KUKA KRL program: Up86.src, Up86.dat

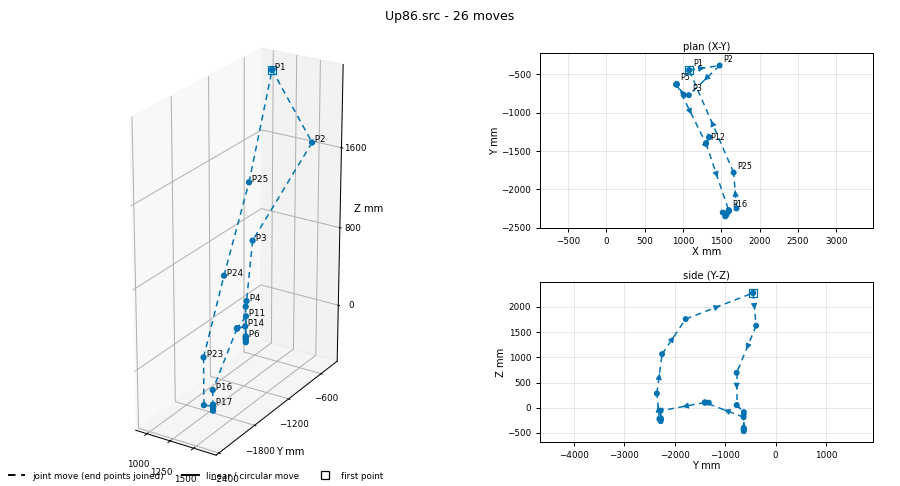
[picture p0: tool path of Up86.src, 26 of 26 moves have a stored position in this frame; points joined in program order, loops and branches not executed]
--- Up86.src ---
&ACCESS RVP
&REL 328
&COMMENT Abdocken 380 Andocken 379
&PARAM DISKPATH = KRC:\R1\UPs
&PARAM TEMPLATE = C:\KRC\Roboter\Template\upvorgabe
&PARAM EDITMASK = Up999[1-999]
&PARAM TPVW_VERSION = 8.1.8
DEF UP86()
   ; FOLD UP Anfang;%{SE} %MKUKATPVW
   SPS_N=-1
   SPS_FERTIG=FALSE
   IF NOT CALLBYSELECT THEN
      INTERRUPT DECL 10 WHEN $CYCFLAG[254]==FALSE DO VW(#FB_STOP,TRUE)
      INTERRUPT ON 10
      INT10=TRUE
      VW_USR_R (#USR_INIT)
   ENDIF
   VW(#VW_INIT_UP,TRUE)
   ; ENDFOLD
   ;FOLD -- TUHR Roboter 5475R01 -- ;%{PSE}%MKUKATPVW,%CVW_COM,%VCOMMENT,%P 1:Comment:, 2:TUHR Roboter 5475R01
      ;FOLD {H}
         M_COMMENT("TUHR Roboter 5475R01")
      ;ENDFOLD
   ;ENDFOLD
   ;FOLD -- Abdocken  VW380 Andocken VW379 -- ;%{PSE}%MKUKATPVW,%CVW_COM,%VCOMMENT,%P 1:Comment:, 2:Abdocken  VW380 Andocken VW379
      ;FOLD {H}
         M_COMMENT("Abdocken  VW380 Andocken VW379")
      ;ENDFOLD
   ;ENDFOLD
   ;FOLD -- DB1 Abdeckklappe AUF -- ;%{PSE}%MKUKATPVW,%CVW_COM,%VCOMMENT,%P 1:Comment:, 2:DB1 Abdeckklappe AUF
      ;FOLD {H}
         M_COMMENT("DB1 Abdeckklappe AUF")
      ;ENDFOLD
   ;ENDFOLD
   ;FOLD -- DB2 Abdeckklappe AUF -- ;%{PSE}%MKUKATPVW,%CVW_COM,%VCOMMENT,%P 1:Comment:, 2:DB2 Abdeckklappe AUF
      ;FOLD {H}
         M_COMMENT("DB2 Abdeckklappe AUF")
      ;ENDFOLD
   ;ENDFOLD
   ;FOLD -- Gespert nur 1 Greifer vorhanden -- ;%{PSE}%MKUKATPVW,%CVW_COM,%VCOMMENT,%P 1:Comment:, 2:Gespert nur 1 Greifer vorhanden
      ;FOLD {H}
         M_COMMENT("Gespert nur 1 Greifer vorhanden")
      ;ENDFOLD
   ;ENDFOLD
   ;FOLD PTP VB=100% VE=0% ACC=100% RobWzg=32 Base=0 SPSTrig=0[1/100s] P ;%{P}%MKUKATPVW,%CMOVE8,%VPTP,%P 1:1, 2: VB=, 3:100, 4:%, 5: VE=, 6:0, 7:%, 8: ACC=, 9:100, 10:%, 11: RobWzg=, 12:32, 13: Base=, 14:0, 15: SPSTrig=, 16:0, 17:[1/100s], 18: P, 19:1, 20:-1, 21:1
      ;FOLD 1: FB PSPS = AUS ;%{SE}%MKUKATPVW %CVW_SPS %VFBPSPS %P 2:FB PSPS = AUS,3:FBPSPS
      ;ENDFOLD
      ;FOLD 2: A23 = AUS ;%{SE}%MKUKATPVW %CVW_SPS %VBOASG %P 2:A23 = AUS,3:BOASG
      ;ENDFOLD
      ;FOLD 3: t6 ( EIN ) = 0[1/10Sek] ;%{SE}%MKUKATPVW %CVW_SPS %VTASG %P 2:t6 ( EIN ) = 0[1/10Sek],3:TASG
      ;ENDFOLD
      ;FOLD 4: SPSMAKRO50 = EIN ;%{SE}%MKUKATPVW %CVW_SPS %VMAKRO %P 2:SPSMAKRO50 = EIN,3:MAKRO
      ;ENDFOLD
      ;FOLD 5: SPSMAKRO53 = EIN ;%{SE}%MKUKATPVW %CVW_SPS %VMAKRO %P 2:SPSMAKRO53 = EIN,3:MAKRO
      ;ENDFOLD
      ;FOLD 6: A42 = EIN ;%{SE}%MKUKATPVW %CVW_SPS %VBOASG %P 2:A42 = EIN,3:BOASG
      ;ENDFOLD
      ;FOLD 7: A43 = EIN ;%{SE}%MKUKATPVW %CVW_SPS %VBOASG %P 2:A43 = EIN,3:BOASG
      ;ENDFOLD
      ;FOLD 8: A44 = EIN ;%{SE}%MKUKATPVW %CVW_SPS %VBOASG %P 2:A44 = EIN,3:BOASG
      ;ENDFOLD
      ;FOLD 9: A45 = EIN ;%{SE}%MKUKATPVW %CVW_SPS %VBOASG %P 2:A45 = EIN,3:BOASG
      ;ENDFOLD
      ;FOLD 10: A47 = EIN ;%{SE}%MKUKATPVW %CVW_SPS %VBOASG %P 2:A47 = EIN,3:BOASG
      ;ENDFOLD
      ;FOLD 11: A49 = EIN ;%{SE}%MKUKATPVW %CVW_SPS %VBOASG %P 2:A49 = EIN,3:BOASG
      ;ENDFOLD
      ;FOLD 12: A52 = EIN ;%{SE}%MKUKATPVW %CVW_SPS %VBOASG %P 2:A52 = EIN,3:BOASG
      ;ENDFOLD
      ;FOLD 13: A54 = EIN ;%{SE}%MKUKATPVW %CVW_SPS %VBOASG %P 2:A54 = EIN,3:BOASG
      ;ENDFOLD
      ;FOLD 14: A75 = EIN ;%{SE}%MKUKATPVW %CVW_SPS %VBOASG %P 2:A75 = EIN,3:BOASG
      ;ENDFOLD
      ;FOLD 15: A76 = EIN ;%{SE}%MKUKATPVW %CVW_SPS %VBOASG %P 2:A76 = EIN,3:BOASG
      ;ENDFOLD
      ;FOLD 16: A79 = EIN ;%{SE}%MKUKATPVW %CVW_SPS %VBOASG %P 2:A79 = EIN,3:BOASG
      ;ENDFOLD
      ;FOLD 17: A80 = EIN ;%{SE}%MKUKATPVW %CVW_SPS %VBOASG %P 2:A80 = EIN,3:BOASG
      ;ENDFOLD
      ;FOLD 18: WARTE BIS M13 & M78 & !E16 ;%{SE}%MKUKATPVW %CVW_SPS %VWBOASG %P 2:WARTE BIS M13 & M78 & !E16,3:WBOASG
      ;ENDFOLD
      ;FOLD 19: F1 = EIN ;%{SE}%MKUKATPVW %CVW_SPS %VBOASG %P 2:F1 = EIN,3:BOASG
      ;ENDFOLD
      ;FOLD 20: F2 = EIN ;%{SE}%MKUKATPVW %CVW_SPS %VBOASG %P 2:F2 = EIN,3:BOASG
      ;ENDFOLD
      ;FOLD 21: SPSMAKRO343 = M13 ;%{SE}%MKUKATPVW %CVW_SPS %VMAKRO %P 2:SPSMAKRO343 = M13,3:MAKRO
      ;ENDFOLD
      ;FOLD 22: SPSMAKRO340 = EIN ;%{SE}%MKUKATPVW %CVW_SPS %VMAKRO %P 2:SPSMAKRO340 = EIN,3:MAKRO
      ;ENDFOLD
      ;FOLD 23: WARTE BIS M32 & M34 ;%{SE}%MKUKATPVW %CVW_SPS %VWBOASG %P 2:WARTE BIS M32 & M34,3:WBOASG
      ;ENDFOLD
      ;FOLD 24: SPSMAKRO430 = EIN ;%{SE}%MKUKATPVW %CVW_SPS %VMAKRO %P 2:SPSMAKRO430 = EIN,3:MAKRO
      ;ENDFOLD
      ;FOLD 25: F841 = EIN ;%{SE}%MKUKATPVW %CVW_SPS %VBOASG %P 2:F841 = EIN,3:BOASG
      ;ENDFOLD
      ;FOLD 26: F842 = EIN ;%{SE}%MKUKATPVW %CVW_SPS %VBOASG %P 2:F842 = EIN,3:BOASG
      ;ENDFOLD
      ;FOLD 27: SPSMAKRO432 = EIN ;%{SE}%MKUKATPVW %CVW_SPS %VMAKRO %P 2:SPSMAKRO432 = EIN,3:MAKRO
      ;ENDFOLD
      ;FOLD 28: WARTE BIS E547 & !E548 & E549 & !E550 & E552 ;%{SE}%MKUKATPVW %CVW_SPS %VWBOASG %P 2:WARTE BIS E547 & !E548 & E549 & !E550 & E552,3:WBOASG
      ;ENDFOLD
      ;FOLD 29: WARTE BIS E23 ;%{SE}%MKUKATPVW %CVW_SPS %VWBOASG %P 2:WARTE BIS E23,3:WBOASG
      ;ENDFOLD
      ;FOLD 30: A23 = EIN ;%{SE}%MKUKATPVW %CVW_SPS %VBOASG %P 2:A23 = EIN,3:BOASG
      ;ENDFOLD
      ;FOLD 31: FB PSPS = M30 & M32 & M34 & M78 & M82 & E547 & E549 ;%{SE}%MKUKATPVW %CVW_SPS %VFBPSPS %P 2:FB PSPS = M30 & M32 & M34 & M78 & M82 & E547 & E549,3:FBPSPS
      ;ENDFOLD
      ;FOLD {H}
         VW_MPARA_ACT=P1_D
         Act_P1 = P1
         Act_P2 = P1
         VW(#MPARA,TRUE)
         SPS_FERTIG=FALSE
         TRIGGER WHEN DISTANCE=1 DELAY=0 DO SPS_TRIG(1) PRIO=-1
         PTP P1
         $ADVANCE=1
         WAIT FOR SPS_FERTIG
      ;ENDFOLD
   ;ENDFOLD
   ;FOLD PTP VB=100% VE=100% ACC=100% RobWzg=32 Base=0 SPSTrig=0[1/100s] P ;%{P}%MKUKATPVW,%CMOVE8,%VPTP,%P 1:1, 2: VB=, 3:100, 4:%, 5: VE=, 6:100, 7:%, 8: ACC=, 9:100, 10:%, 11: RobWzg=, 12:32, 13: Base=, 14:0, 15: SPSTrig=, 16:0, 17:[1/100s], 18: P, 19:2, 20:-1, 21:2
      ;FOLD 1: FB PSPS = M30 & M32 & M34 & M78 & M82 & E547 & E549 ;%{SE}%MKUKATPVW %CVW_SPS %VFBPSPS %P 2:FB PSPS = M30 & M32 & M34 & M78 & M82 & E547 & E549,3:FBPSPS
      ;ENDFOLD
      ;FOLD {H}
         VW_MPARA_ACT=P2_D
         Act_P1 = P2
         Act_P2 = P2
         VW(#MPARA,TRUE)
         SPS_FERTIG=FALSE
         TRIGGER WHEN DISTANCE=1 DELAY=0 DO SPS_TRIG(10002) PRIO=-1
         PTP P2 C_PTP C_VEL
         $ADVANCE=1
      ;ENDFOLD
   ;ENDFOLD
   ;FOLD PTP VB=100% VE=100% ACC=100% RobWzg=32 Base=0 SPSTrig=0[1/100s] P ;%{P}%MKUKATPVW,%CMOVE8,%VPTP,%P 1:1, 2: VB=, 3:100, 4:%, 5: VE=, 6:100, 7:%, 8: ACC=, 9:100, 10:%, 11: RobWzg=, 12:32, 13: Base=, 14:0, 15: SPSTrig=, 16:0, 17:[1/100s], 18: P, 19:3, 20:-1, 21:3
      ;FOLD 1: FB PSPS = M30 & M32 & M34 & M78 & M82 & E547 & E549 ;%{SE}%MKUKATPVW %CVW_SPS %VFBPSPS %P 2:FB PSPS = M30 & M32 & M34 & M78 & M82 & E547 & E549,3:FBPSPS
      ;ENDFOLD
      ;FOLD {H}
         VW_MPARA_ACT=P3_D
         Act_P1 = P3
         Act_P2 = P3
         VW(#MPARA,TRUE)
         SPS_FERTIG=FALSE
         TRIGGER WHEN DISTANCE=1 DELAY=0 DO SPS_TRIG(10003) PRIO=-1
         PTP P3 C_PTP C_VEL
         $ADVANCE=1
      ;ENDFOLD
   ;ENDFOLD
   ;FOLD PTP VB=100% VE=100% ACC=100% RobWzg=32 Base=0 SPSTrig=0[1/100s] P ;%{P}%MKUKATPVW,%CMOVE8,%VPTP,%P 1:1, 2: VB=, 3:100, 4:%, 5: VE=, 6:100, 7:%, 8: ACC=, 9:100, 10:%, 11: RobWzg=, 12:32, 13: Base=, 14:0, 15: SPSTrig=, 16:0, 17:[1/100s], 18: P, 19:4, 20:-1, 21:4
      ;FOLD 1: FB PSPS = M30 & M32 & M34 & M78 & M82 & E547 & E549 ;%{SE}%MKUKATPVW %CVW_SPS %VFBPSPS %P 2:FB PSPS = M30 & M32 & M34 & M78 & M82 & E547 & E549,3:FBPSPS
      ;ENDFOLD
      ;FOLD {H}
         VW_MPARA_ACT=P4_D
         Act_P1 = P4
         Act_P2 = P4
         VW(#MPARA,TRUE)
         SPS_FERTIG=FALSE
         TRIGGER WHEN DISTANCE=1 DELAY=0 DO SPS_TRIG(10004) PRIO=-1
         PTP P4 C_PTP C_VEL
         $ADVANCE=1
      ;ENDFOLD
   ;ENDFOLD
   ;FOLD PTP VB=100% VE=100% ACC=100% RobWzg=32 Base=0 SPSTrig=0[1/100s] P ;%{P}%MKUKATPVW,%CMOVE8,%VPTP,%P 1:1, 2: VB=, 3:100, 4:%, 5: VE=, 6:100, 7:%, 8: ACC=, 9:100, 10:%, 11: RobWzg=, 12:32, 13: Base=, 14:0, 15: SPSTrig=, 16:0, 17:[1/100s], 18: P, 19:5, 20:-1, 21:5
      ;FOLD 1: FB PSPS = M30 & M32 & M34 & M78 & M82 & E547 & E549 ;%{SE}%MKUKATPVW %CVW_SPS %VFBPSPS %P 2:FB PSPS = M30 & M32 & M34 & M78 & M82 & E547 & E549,3:FBPSPS
      ;ENDFOLD
      ;FOLD {H}
         VW_MPARA_ACT=P5_D
         Act_P1 = P5
         Act_P2 = P5
         VW(#MPARA,TRUE)
         SPS_FERTIG=FALSE
         TRIGGER WHEN DISTANCE=1 DELAY=0 DO SPS_TRIG(10005) PRIO=-1
         PTP P5 C_PTP C_VEL
         $ADVANCE=1
      ;ENDFOLD
   ;ENDFOLD
   ;FOLD -- Profinet  Teilnehmer  abschalten -- ;%{PSE}%MKUKATPVW,%CVW_COM,%VCOMMENT,%P 1:Comment:, 2:Profinet  Teilnehmer  abschalten
      ;FOLD {H}
         M_COMMENT("Profinet  Teilnehmer  abschalten")
      ;ENDFOLD
   ;ENDFOLD
   ;FOLD PTP VB=100% VE=0% ACC=100% RobWzg=32 Base=0 SPSTrig=0[1/100s] P ;%{P}%MKUKATPVW,%CMOVE8,%VPTP,%P 1:1, 2: VB=, 3:100, 4:%, 5: VE=, 6:0, 7:%, 8: ACC=, 9:100, 10:%, 11: RobWzg=, 12:32, 13: Base=, 14:0, 15: SPSTrig=, 16:0, 17:[1/100s], 18: P, 19:6, 20:-1, 21:6
      ;FOLD 1: FB PSPS = EIN ;%{SE}%MKUKATPVW %CVW_SPS %VFBPSPS %P 2:FB PSPS = EIN,3:FBPSPS
      ;ENDFOLD
      ;FOLD 2: A23 = AUS ;%{SE}%MKUKATPVW %CVW_SPS %VBOASG %P 2:A23 = AUS,3:BOASG
      ;ENDFOLD
      ;FOLD 3: SPSMAKRO422 = !E540 ;%{SE}%MKUKATPVW %CVW_SPS %VMAKRO %P 2:SPSMAKRO422 = !E540,3:MAKRO
      ;ENDFOLD
      ;FOLD 4: WARTE BIS E540 & !E551 & E23 ;%{SE}%MKUKATPVW %CVW_SPS %VWBOASG %P 2:WARTE BIS E540 & !E551 & E23,3:WBOASG
      ;ENDFOLD
      ;FOLD 5: TECH3_ PN-Docken ID-Nr =122 Abschalten EIN ;%{SE}%MKUKATPVW %CVW_SPS %VUSER %P 2:TECH3_.PN-Docken P1= 122 P2= 60 P3= 1 P4= 1 P5= 1 P6= 1 P7=EIN P8=301,3:USER
      ;ENDFOLD
      ;FOLD 6: A23 = EIN ;%{SE}%MKUKATPVW %CVW_SPS %VBOASG %P 2:A23 = EIN,3:BOASG
      ;ENDFOLD
      ;FOLD 7: FB PSPS = M30 & M78 & E547 & E549 ;%{SE}%MKUKATPVW %CVW_SPS %VFBPSPS %P 2:FB PSPS = M30 & M78 & E547 & E549,3:FBPSPS
      ;ENDFOLD
      ;FOLD {H}
         VW_MPARA_ACT=P6_D
         Act_P1 = P6
         Act_P2 = P6
         VW(#MPARA,TRUE)
         SPS_FERTIG=FALSE
         TRIGGER WHEN DISTANCE=1 DELAY=0 DO SPS_TRIG(6) PRIO=-1
         VW_USER (#USR_ADV,301,122,60,1,1,1,1,TRUE)
         VW_USR_R (#USR_ADV,301,122,60,1,1,1,1,TRUE)
         PTP P6
         $ADVANCE=1
         WAIT FOR SPS_FERTIG
         VW_USER (#USR_MAIN,301,122,60,1,1,1,1,TRUE)
         VW_USR_R (#USR_MAIN,301,122,60,1,1,1,1,TRUE)
      ;ENDFOLD
   ;ENDFOLD
   ;FOLD -- Ueber  DB -- ;%{PSE}%MKUKATPVW,%CVW_COM,%VCOMMENT,%P 1:Comment:, 2:Ueber  DB
      ;FOLD {H}
         M_COMMENT("Ueber  DB")
      ;ENDFOLD
   ;ENDFOLD
   ;FOLD LIN VB=200[mm/s] VE=0% ACC=100% RobWzg=32 Base=0 SPSTrig=5[1/100s] P ;%{P}%MKUKATPVW,%CMOVE8,%VLIN,%P 1:2, 2: VB=, 3:200, 4:[mm/s], 5: VE=, 6:0, 7:%, 8: ACC=, 9:100, 10:%, 11: RobWzg=, 12:32, 13: Base=, 14:0, 15: SPSTrig=, 16:5, 17:[1/100s], 18: P, 19:7, 20:-1, 21:7
      ;FOLD 1: FB PSPS = M30 & M78 & E547 & E549 ;%{SE}%MKUKATPVW %CVW_SPS %VFBPSPS %P 2:FB PSPS = M30 & M78 & E547 & E549,3:FBPSPS
      ;ENDFOLD
      ;FOLD {H}
         VW_MPARA_ACT=P7_D
         Act_P1 = P7
         Act_P2 = P7
         VW(#MPARA,TRUE)
         SPS_FERTIG=FALSE
         TRIGGER WHEN DISTANCE=1 DELAY=-50 DO SPS_TRIG(7) PRIO=-1
         LIN P7
         $ADVANCE=1
         WAIT FOR SPS_FERTIG
      ;ENDFOLD
   ;ENDFOLD
   ;FOLD -- Abdockposition VW380 4T 5425r01 -- ;%{PSE}%MKUKATPVW,%CVW_COM,%VCOMMENT,%P 1:Comment:, 2:Abdockposition VW380 4T 5425r01
      ;FOLD {H}
         M_COMMENT("Abdockposition VW380 4T 5425r01")
      ;ENDFOLD
   ;ENDFOLD
   ;FOLD LIN VB=50[mm/s] VE=0% ACC=100% RobWzg=32 Base=0 SPSTrig=5[1/100s] P ;%{P}%MKUKATPVW,%CMOVE8,%VLIN,%P 1:2, 2: VB=, 3:50, 4:[mm/s], 5: VE=, 6:0, 7:%, 8: ACC=, 9:100, 10:%, 11: RobWzg=, 12:32, 13: Base=, 14:0, 15: SPSTrig=, 16:5, 17:[1/100s], 18: P, 19:8, 20:-1, 21:8
      ;FOLD 1: FB PSPS = EIN ;%{SE}%MKUKATPVW %CVW_SPS %VFBPSPS %P 2:FB PSPS = EIN,3:FBPSPS
      ;ENDFOLD
      ;FOLD 2: A23 = AUS ;%{SE}%MKUKATPVW %CVW_SPS %VBOASG %P 2:A23 = AUS,3:BOASG
      ;ENDFOLD
      ;FOLD 3: WARTE BIS E540 & E551 & E23 ;%{SE}%MKUKATPVW %CVW_SPS %VWBOASG %P 2:WARTE BIS E540 & E551 & E23,3:WBOASG
      ;ENDFOLD
      ;FOLD 4: A23 = EIN ;%{SE}%MKUKATPVW %CVW_SPS %VBOASG %P 2:A23 = EIN,3:BOASG
      ;ENDFOLD
      ;FOLD 5: SPSMAKRO420 = EIN ;%{SE}%MKUKATPVW %CVW_SPS %VMAKRO %P 2:SPSMAKRO420 = EIN,3:MAKRO
      ;ENDFOLD
      ;FOLD 6: WARTE BIS !E538 & E539 ;%{SE}%MKUKATPVW %CVW_SPS %VWBOASG %P 2:WARTE BIS !E538 & E539,3:WBOASG
      ;ENDFOLD
      ;FOLD 7: FB PSPS = M30 & !E538 & E539 & E540 & E551 & E552 ;%{SE}%MKUKATPVW %CVW_SPS %VFBPSPS %P 2:FB PSPS = M30 & !E538 & E539 & E540 & E551 & E552,3:FBPSPS
      ;ENDFOLD
      ;FOLD {H}
         VW_MPARA_ACT=P8_D
         Act_P1 = P8
         Act_P2 = P8
         VW(#MPARA,TRUE)
         SPS_FERTIG=FALSE
         TRIGGER WHEN DISTANCE=1 DELAY=-50 DO SPS_TRIG(8) PRIO=-1
         LIN P8
         $ADVANCE=1
         WAIT FOR SPS_FERTIG
      ;ENDFOLD
   ;ENDFOLD
   ;FOLD -- Ueber  DB1  WASI  noch  belegt -- ;%{PSE}%MKUKATPVW,%CVW_COM,%VCOMMENT,%P 1:Comment:, 2:Ueber  DB1  WASI  noch  belegt
      ;FOLD {H}
         M_COMMENT("Ueber  DB1  WASI  noch  belegt")
      ;ENDFOLD
   ;ENDFOLD
   ;FOLD LIN VB=50[mm/s] VE=10% ACC=100% RobWzg=32 Base=0 SPSTrig=5[1/100s] P ;%{P}%MKUKATPVW,%CMOVE8,%VLIN,%P 1:2, 2: VB=, 3:50, 4:[mm/s], 5: VE=, 6:10, 7:%, 8: ACC=, 9:100, 10:%, 11: RobWzg=, 12:32, 13: Base=, 14:0, 15: SPSTrig=, 16:5, 17:[1/100s], 18: P, 19:9, 20:-1, 21:9
      ;FOLD 1: FB PSPS = M30 & E547 & E549 & E551 & E552 ;%{SE}%MKUKATPVW %CVW_SPS %VFBPSPS %P 2:FB PSPS = M30 & E547 & E549 & E551 & E552,3:FBPSPS
      ;ENDFOLD
      ;FOLD {H}
         VW_MPARA_ACT=P9_D
         Act_P1 = P9
         Act_P2 = P9
         VW(#MPARA,TRUE)
         SPS_FERTIG=FALSE
         TRIGGER WHEN DISTANCE=1 DELAY=-50 DO SPS_TRIG(10009) PRIO=-1
         LIN P9 C_VEL
         $ADVANCE=1
      ;ENDFOLD
   ;ENDFOLD
   ;FOLD -- Ueber  DB1 -- ;%{PSE}%MKUKATPVW,%CVW_COM,%VCOMMENT,%P 1:Comment:, 2:Ueber  DB1
      ;FOLD {H}
         M_COMMENT("Ueber  DB1")
      ;ENDFOLD
   ;ENDFOLD
   ;FOLD LIN VB=100[mm/s] VE=50% ACC=100% RobWzg=32 Base=0 SPSTrig=0[1/100s] P ;%{P}%MKUKATPVW,%CMOVE8,%VLIN,%P 1:2, 2: VB=, 3:100, 4:[mm/s], 5: VE=, 6:50, 7:%, 8: ACC=, 9:100, 10:%, 11: RobWzg=, 12:32, 13: Base=, 14:0, 15: SPSTrig=, 16:0, 17:[1/100s], 18: P, 19:10, 20:-1, 21:10
      ;FOLD 1: FB PSPS = EIN ;%{SE}%MKUKATPVW %CVW_SPS %VFBPSPS %P 2:FB PSPS = EIN,3:FBPSPS
      ;ENDFOLD
      ;FOLD 2: A539 = AUS ;%{SE}%MKUKATPVW %CVW_SPS %VBOASG %P 2:A539 = AUS,3:BOASG
      ;ENDFOLD
      ;FOLD 3: FB PSPS = M30 & E547 & E549 & E551 & E552 ;%{SE}%MKUKATPVW %CVW_SPS %VFBPSPS %P 2:FB PSPS = M30 & E547 & E549 & E551 & E552,3:FBPSPS
      ;ENDFOLD
      ;FOLD {H}
         VW_MPARA_ACT=P10_D
         Act_P1 = P10
         Act_P2 = P10
         VW(#MPARA,TRUE)
         SPS_FERTIG=FALSE
         TRIGGER WHEN DISTANCE=1 DELAY=0 DO SPS_TRIG(10010) PRIO=-1
         LIN P10 C_VEL
         $ADVANCE=1
      ;ENDFOLD
   ;ENDFOLD
   ;FOLD PTP VB=100% VE=100% ACC=100% RobWzg=32 Base=0 SPSTrig=0[1/100s] P ;%{P}%MKUKATPVW,%CMOVE8,%VPTP,%P 1:1, 2: VB=, 3:100, 4:%, 5: VE=, 6:100, 7:%, 8: ACC=, 9:100, 10:%, 11: RobWzg=, 12:32, 13: Base=, 14:0, 15: SPSTrig=, 16:0, 17:[1/100s], 18: P, 19:11, 20:-1, 21:11
      ;FOLD 1: FB PSPS = M30 & E547 & E549 & E551 & E552 ;%{SE}%MKUKATPVW %CVW_SPS %VFBPSPS %P 2:FB PSPS = M30 & E547 & E549 & E551 & E552,3:FBPSPS
      ;ENDFOLD
      ;FOLD {H}
         VW_MPARA_ACT=P11_D
         Act_P1 = P11
         Act_P2 = P11
         VW(#MPARA,TRUE)
         SPS_FERTIG=FALSE
         TRIGGER WHEN DISTANCE=1 DELAY=0 DO SPS_TRIG(10011) PRIO=-1
         PTP P11 C_PTP C_VEL
         $ADVANCE=1
      ;ENDFOLD
   ;ENDFOLD
   ;FOLD PTP VB=100% VE=100% ACC=100% RobWzg=32 Base=0 SPSTrig=0[1/100s] P ;%{P}%MKUKATPVW,%CMOVE8,%VPTP,%P 1:1, 2: VB=, 3:100, 4:%, 5: VE=, 6:100, 7:%, 8: ACC=, 9:100, 10:%, 11: RobWzg=, 12:32, 13: Base=, 14:0, 15: SPSTrig=, 16:0, 17:[1/100s], 18: P, 19:12, 20:-1, 21:12
      ;FOLD 1: FB PSPS = M30 & E547 & E549 & E551 & E552 ;%{SE}%MKUKATPVW %CVW_SPS %VFBPSPS %P 2:FB PSPS = M30 & E547 & E549 & E551 & E552,3:FBPSPS
      ;ENDFOLD
      ;FOLD {H}
         VW_MPARA_ACT=P12_D
         Act_P1 = P12
         Act_P2 = P12
         VW(#MPARA,TRUE)
         SPS_FERTIG=FALSE
         TRIGGER WHEN DISTANCE=1 DELAY=0 DO SPS_TRIG(10012) PRIO=-1
         PTP P12 C_PTP C_VEL
         $ADVANCE=1
      ;ENDFOLD
   ;ENDFOLD
   ;FOLD PTP VB=100% VE=0% ACC=100% RobWzg=32 Base=0 SPSTrig=0[1/100s] P ;%{P}%MKUKATPVW,%CMOVE8,%VPTP,%P 1:1, 2: VB=, 3:100, 4:%, 5: VE=, 6:0, 7:%, 8: ACC=, 9:100, 10:%, 11: RobWzg=, 12:32, 13: Base=, 14:0, 15: SPSTrig=, 16:0, 17:[1/100s], 18: P, 19:13, 20:-1, 21:13
      ;FOLD 1: FB PSPS = EIN ;%{SE}%MKUKATPVW %CVW_SPS %VFBPSPS %P 2:FB PSPS = EIN,3:FBPSPS
      ;ENDFOLD
      ;FOLD 2: F842 = EIN ;%{SE}%MKUKATPVW %CVW_SPS %VBOASG %P 2:F842 = EIN,3:BOASG
      ;ENDFOLD
      ;FOLD 3: SPSMAKRO433 = EIN ;%{SE}%MKUKATPVW %CVW_SPS %VMAKRO %P 2:SPSMAKRO433 = EIN,3:MAKRO
      ;ENDFOLD
      ;FOLD 4: F841 = EIN ;%{SE}%MKUKATPVW %CVW_SPS %VBOASG %P 2:F841 = EIN,3:BOASG
      ;ENDFOLD
      ;FOLD 5: SPSMAKRO432 = EIN ;%{SE}%MKUKATPVW %CVW_SPS %VMAKRO %P 2:SPSMAKRO432 = EIN,3:MAKRO
      ;ENDFOLD
      ;FOLD 6: WARTE BIS E549 & !E550 & E23 ;%{SE}%MKUKATPVW %CVW_SPS %VWBOASG %P 2:WARTE BIS E549 & !E550 & E23,3:WBOASG
      ;ENDFOLD
      ;FOLD 7: A539 = AUS ;%{SE}%MKUKATPVW %CVW_SPS %VBOASG %P 2:A539 = AUS,3:BOASG
      ;ENDFOLD
      ;FOLD 8: A23 = AUS ;%{SE}%MKUKATPVW %CVW_SPS %VBOASG %P 2:A23 = AUS,3:BOASG
      ;ENDFOLD
      ;FOLD 9: WARTE BIS E23 ;%{SE}%MKUKATPVW %CVW_SPS %VWBOASG %P 2:WARTE BIS E23,3:WBOASG
      ;ENDFOLD
      ;FOLD 10: A23 = EIN ;%{SE}%MKUKATPVW %CVW_SPS %VBOASG %P 2:A23 = EIN,3:BOASG
      ;ENDFOLD
      ;FOLD 11: F958 = !F933 ;%{SE}%MKUKATPVW %CVW_SPS %VBOASG %P 2:F958 = !F933,3:BOASG
      ;ENDFOLD
      ;FOLD 12: FB PSPS = M30 & !E547 & E548 & E549 & E551 & E552 ;%{SE}%MKUKATPVW %CVW_SPS %VFBPSPS %P 2:FB PSPS = M30 & !E547 & E548 & E549 & E551 & E552,3:FBPSPS
      ;ENDFOLD
      ;FOLD {H}
         VW_MPARA_ACT=P13_D
         Act_P1 = P13
         Act_P2 = P13
         VW(#MPARA,TRUE)
         SPS_FERTIG=FALSE
         TRIGGER WHEN DISTANCE=1 DELAY=0 DO SPS_TRIG(13) PRIO=-1
         PTP P13
         $ADVANCE=1
         WAIT FOR SPS_FERTIG
      ;ENDFOLD
   ;ENDFOLD
   ;FOLD GOTO Label 1 = F958 ;%{PSE}%MKUKATPVW,%CCONTROL,%VJUMP,%P 1:GOTO Label, 2:1, 3:=, 4:6, 5:958
      ;FOLD  ;%{H}
         CONTINUE
         IF $FLAG[958] THEN
            CONTINUE
            GOTO Label1
         ENDIF
      ;ENDFOLD
   ;ENDFOLD
   ;FOLD -- Wartung  Dockingklappe -- ;%{PSE}%MKUKATPVW,%CVW_COM,%VCOMMENT,%P 1:Comment:, 2:Wartung  Dockingklappe
      ;FOLD {H}
         M_COMMENT("Wartung  Dockingklappe")
      ;ENDFOLD
   ;ENDFOLD
   ;FOLD PTP VB=100% VE=0% ACC=100% RobWzg=32 Base=0 SPSTrig=0[1/100s] P ;%{P}%MKUKATPVW,%CMOVE8,%VPTP,%P 1:1, 2: VB=, 3:100, 4:%, 5: VE=, 6:0, 7:%, 8: ACC=, 9:100, 10:%, 11: RobWzg=, 12:32, 13: Base=, 14:0, 15: SPSTrig=, 16:0, 17:[1/100s], 18: P, 19:14, 20:-1, 21:14
      ;FOLD 1: FB PSPS = EIN ;%{SE}%MKUKATPVW %CVW_SPS %VFBPSPS %P 2:FB PSPS = EIN,3:FBPSPS
      ;ENDFOLD
      ;FOLD 2: A23 = AUS ;%{SE}%MKUKATPVW %CVW_SPS %VBOASG %P 2:A23 = AUS,3:BOASG
      ;ENDFOLD
      ;FOLD 3: F841 = EIN ;%{SE}%MKUKATPVW %CVW_SPS %VBOASG %P 2:F841 = EIN,3:BOASG
      ;ENDFOLD
      ;FOLD 4: F842 = EIN ;%{SE}%MKUKATPVW %CVW_SPS %VBOASG %P 2:F842 = EIN,3:BOASG
      ;ENDFOLD
      ;FOLD 5: SPSMAKRO433 = EIN ;%{SE}%MKUKATPVW %CVW_SPS %VMAKRO %P 2:SPSMAKRO433 = EIN,3:MAKRO
      ;ENDFOLD
      ;FOLD 6: WARTE BIS !E549 & E550 & !E547 & E548 & E23 ;%{SE}%MKUKATPVW %CVW_SPS %VWBOASG %P 2:WARTE BIS !E549 & E550 & !E547 & E548 & E23,3:WBOASG
      ;ENDFOLD
      ;FOLD 7: SPSMAKRO430 = EIN ;%{SE}%MKUKATPVW %CVW_SPS %VMAKRO %P 2:SPSMAKRO430 = EIN,3:MAKRO
      ;ENDFOLD
      ;FOLD 8: A17 = EIN ;%{SE}%MKUKATPVW %CVW_SPS %VBOASG %P 2:A17 = EIN,3:BOASG
      ;ENDFOLD
      ;FOLD 9: bin19 ( EIN ) = 0 ;%{SE}%MKUKATPVW %CVW_SPS %VARIASG %P 2:bin19 ( EIN ) = 0,3:ARIASG
      ;ENDFOLD
      ;FOLD 10: WARTE BIS E17 ;%{SE}%MKUKATPVW %CVW_SPS %VWBOASG %P 2:WARTE BIS E17,3:WBOASG
      ;ENDFOLD
      ;FOLD 11: A17 = AUS ;%{SE}%MKUKATPVW %CVW_SPS %VBOASG %P 2:A17 = AUS,3:BOASG
      ;ENDFOLD
      ;FOLD 12: F933 = AUS ;%{SE}%MKUKATPVW %CVW_SPS %VBOASG %P 2:F933 = AUS,3:BOASG
      ;ENDFOLD
      ;FOLD 13: F958 = AUS ;%{SE}%MKUKATPVW %CVW_SPS %VBOASG %P 2:F958 = AUS,3:BOASG
      ;ENDFOLD
      ;FOLD 14: F841 = EIN ;%{SE}%MKUKATPVW %CVW_SPS %VBOASG %P 2:F841 = EIN,3:BOASG
      ;ENDFOLD
      ;FOLD 15: SPSMAKRO432 = EIN ;%{SE}%MKUKATPVW %CVW_SPS %VMAKRO %P 2:SPSMAKRO432 = EIN,3:MAKRO
      ;ENDFOLD
      ;FOLD 16: WARTE BIS E549 & !E550 ;%{SE}%MKUKATPVW %CVW_SPS %VWBOASG %P 2:WARTE BIS E549 & !E550,3:WBOASG
      ;ENDFOLD
      ;FOLD 17: WARTE BIS E23 ;%{SE}%MKUKATPVW %CVW_SPS %VWBOASG %P 2:WARTE BIS E23,3:WBOASG
      ;ENDFOLD
      ;FOLD 18: A23 = EIN ;%{SE}%MKUKATPVW %CVW_SPS %VBOASG %P 2:A23 = EIN,3:BOASG
      ;ENDFOLD
      ;FOLD 19: FB PSPS = M30 & !E547 & E548 & E549 & E551 & E552 ;%{SE}%MKUKATPVW %CVW_SPS %VFBPSPS %P 2:FB PSPS = M30 & !E547 & E548 & E549 & E551 & E552,3:FBPSPS
      ;ENDFOLD
      ;FOLD {H}
         VW_MPARA_ACT=P14_D
         Act_P1 = P14
         Act_P2 = P14
         VW(#MPARA,TRUE)
         SPS_FERTIG=FALSE
         TRIGGER WHEN DISTANCE=1 DELAY=0 DO SPS_TRIG(14) PRIO=-1
         PTP P14
         $ADVANCE=1
         WAIT FOR SPS_FERTIG
      ;ENDFOLD
   ;ENDFOLD
   ;FOLD Label 1 ;%{PSE}%MKUKATPVW,%CCONTROL,%VLABEL,%P 1:Label, 2:Label 1
      ;FOLD  ;%{H}
         Label1:
      ;ENDFOLD
   ;ENDFOLD
   ;FOLD PTP VB=100% VE=0% ACC=100% RobWzg=32 Base=0 SPSTrig=0[1/100s] P ;%{P}%MKUKATPVW,%CMOVE8,%VPTP,%P 1:1, 2: VB=, 3:100, 4:%, 5: VE=, 6:0, 7:%, 8: ACC=, 9:100, 10:%, 11: RobWzg=, 12:32, 13: Base=, 14:0, 15: SPSTrig=, 16:0, 17:[1/100s], 18: P, 19:15, 20:-1, 21:15
      ;FOLD 1: FB PSPS = EIN ;%{SE}%MKUKATPVW %CVW_SPS %VFBPSPS %P 2:FB PSPS = EIN,3:FBPSPS
      ;ENDFOLD
      ;FOLD 2: A23 = AUS ;%{SE}%MKUKATPVW %CVW_SPS %VBOASG %P 2:A23 = AUS,3:BOASG
      ;ENDFOLD
      ;FOLD 3: SPSMAKRO422 = !E540 ;%{SE}%MKUKATPVW %CVW_SPS %VMAKRO %P 2:SPSMAKRO422 = !E540,3:MAKRO
      ;ENDFOLD
      ;FOLD 4: WARTE BIS E540 & E23 ;%{SE}%MKUKATPVW %CVW_SPS %VWBOASG %P 2:WARTE BIS E540 & E23,3:WBOASG
      ;ENDFOLD
      ;FOLD 5: A23 = EIN ;%{SE}%MKUKATPVW %CVW_SPS %VBOASG %P 2:A23 = EIN,3:BOASG
      ;ENDFOLD
      ;FOLD 6: FB PSPS = M30 & !E547 & E548 & E549 & E551 & E552 ;%{SE}%MKUKATPVW %CVW_SPS %VFBPSPS %P 2:FB PSPS = M30 & !E547 & E548 & E549 & E551 & E552,3:FBPSPS
      ;ENDFOLD
      ;FOLD {H}
         VW_MPARA_ACT=P15_D
         Act_P1 = P15
         Act_P2 = P15
         VW(#MPARA,TRUE)
         SPS_FERTIG=FALSE
         TRIGGER WHEN DISTANCE=1 DELAY=0 DO SPS_TRIG(15) PRIO=-1
         PTP P15
         $ADVANCE=1
         WAIT FOR SPS_FERTIG
      ;ENDFOLD
   ;ENDFOLD
   ;FOLD PTP VB=100% VE=100% ACC=100% RobWzg=32 Base=0 SPSTrig=0[1/100s] P ;%{P}%MKUKATPVW,%CMOVE8,%VPTP,%P 1:1, 2: VB=, 3:100, 4:%, 5: VE=, 6:100, 7:%, 8: ACC=, 9:100, 10:%, 11: RobWzg=, 12:32, 13: Base=, 14:0, 15: SPSTrig=, 16:0, 17:[1/100s], 18: P, 19:16, 20:-1, 21:16
      ;FOLD 1: FB PSPS = M30 & !E547 & E548 & E549 & E551 & E552 ;%{SE}%MKUKATPVW %CVW_SPS %VFBPSPS %P 2:FB PSPS = M30 & !E547 & E548 & E549 & E551 & E552,3:FBPSPS
      ;ENDFOLD
      ;FOLD {H}
         VW_MPARA_ACT=P16_D
         Act_P1 = P16
         Act_P2 = P16
         VW(#MPARA,TRUE)
         SPS_FERTIG=FALSE
         TRIGGER WHEN DISTANCE=1 DELAY=0 DO SPS_TRIG(10016) PRIO=-1
         PTP P16 C_PTP C_VEL
         $ADVANCE=1
      ;ENDFOLD
   ;ENDFOLD
   ;FOLD PTP VB=100% VE=100% ACC=100% RobWzg=32 Base=0 SPSTrig=0[1/100s] P ;%{P}%MKUKATPVW,%CMOVE8,%VPTP,%P 1:1, 2: VB=, 3:100, 4:%, 5: VE=, 6:100, 7:%, 8: ACC=, 9:100, 10:%, 11: RobWzg=, 12:32, 13: Base=, 14:0, 15: SPSTrig=, 16:0, 17:[1/100s], 18: P, 19:17, 20:-1, 21:17
      ;FOLD 1: FB PSPS = M30 & !E547 & E548 & E549 & E551 & E552 ;%{SE}%MKUKATPVW %CVW_SPS %VFBPSPS %P 2:FB PSPS = M30 & !E547 & E548 & E549 & E551 & E552,3:FBPSPS
      ;ENDFOLD
      ;FOLD {H}
         VW_MPARA_ACT=P17_D
         Act_P1 = P17
         Act_P2 = P17
         VW(#MPARA,TRUE)
         SPS_FERTIG=FALSE
         TRIGGER WHEN DISTANCE=1 DELAY=0 DO SPS_TRIG(10017) PRIO=-1
         PTP P17 C_PTP C_VEL
         $ADVANCE=1
      ;ENDFOLD
   ;ENDFOLD
   ;FOLD -- Dockingsystem Entriegeln -- ;%{PSE}%MKUKATPVW,%CVW_COM,%VCOMMENT,%P 1:Comment:, 2:Dockingsystem Entriegeln
      ;FOLD {H}
         M_COMMENT("Dockingsystem Entriegeln")
      ;ENDFOLD
   ;ENDFOLD
   ;FOLD LIN VB=300[mm/s] VE=0% ACC=100% RobWzg=32 Base=0 SPSTrig=5[1/100s] P ;%{P}%MKUKATPVW,%CMOVE8,%VLIN,%P 1:2, 2: VB=, 3:300, 4:[mm/s], 5: VE=, 6:0, 7:%, 8: ACC=, 9:100, 10:%, 11: RobWzg=, 12:32, 13: Base=, 14:0, 15: SPSTrig=, 16:5, 17:[1/100s], 18: P, 19:18, 20:-1, 21:18
      ;FOLD 1: FB PSPS = EIN ;%{SE}%MKUKATPVW %CVW_SPS %VFBPSPS %P 2:FB PSPS = EIN,3:FBPSPS
      ;ENDFOLD
      ;FOLD 2: A23 = AUS ;%{SE}%MKUKATPVW %CVW_SPS %VBOASG %P 2:A23 = AUS,3:BOASG
      ;ENDFOLD
      ;FOLD 3: WARTE BIS E23 ;%{SE}%MKUKATPVW %CVW_SPS %VWBOASG %P 2:WARTE BIS E23,3:WBOASG
      ;ENDFOLD
      ;FOLD 4: A23 = EIN ;%{SE}%MKUKATPVW %CVW_SPS %VBOASG %P 2:A23 = EIN,3:BOASG
      ;ENDFOLD
      ;FOLD 5: SPSMAKRO52 = EIN ;%{SE}%MKUKATPVW %CVW_SPS %VMAKRO %P 2:SPSMAKRO52 = EIN,3:MAKRO
      ;ENDFOLD
      ;FOLD 6: -- DK Entriegeln -- ;%{SE}%MKUKATPVW %CVW_COM %VCOMMENT %P 2:-- DK Entriegeln --,3:VW_COMMENT
      ;ENDFOLD
      ;FOLD 7: A539 = EIN ;%{SE}%MKUKATPVW %CVW_SPS %VBOASG %P 2:A539 = EIN,3:BOASG
      ;ENDFOLD
      ;FOLD 8: WARTE BIS !E538 & E539 & E540 ;%{SE}%MKUKATPVW %CVW_SPS %VWBOASG %P 2:WARTE BIS !E538 & E539 & E540,3:WBOASG
      ;ENDFOLD
      ;FOLD 9: FB PSPS = M30 & !E538 & E539 & E548 & E549 & E551 & E552 ;%{SE}%MKUKATPVW %CVW_SPS %VFBPSPS %P 2:FB PSPS = M30 & !E538 & E539 & E548 & E549 & E551 & E552,3:FBPSPS
      ;ENDFOLD
      ;FOLD {H}
         VW_MPARA_ACT=P18_D
         Act_P1 = P18
         Act_P2 = P18
         VW(#MPARA,TRUE)
         SPS_FERTIG=FALSE
         TRIGGER WHEN DISTANCE=1 DELAY=-50 DO SPS_TRIG(18) PRIO=-1
         LIN P18
         $ADVANCE=1
         WAIT FOR SPS_FERTIG
      ;ENDFOLD
   ;ENDFOLD
   ;FOLD -- Andockposition VW310 4525r01 -- ;%{PSE}%MKUKATPVW,%CVW_COM,%VCOMMENT,%P 1:Comment:, 2:Andockposition VW310 4525r01
      ;FOLD {H}
         M_COMMENT("Andockposition VW310 4525r01")
      ;ENDFOLD
   ;ENDFOLD
   ;FOLD LIN VB=100[mm/s] VE=0% ACC=100% RobWzg=32 Base=0 SPSTrig=5[1/100s] P ;%{P}%MKUKATPVW,%CMOVE8,%VLIN,%P 1:2, 2: VB=, 3:100, 4:[mm/s], 5: VE=, 6:0, 7:%, 8: ACC=, 9:100, 10:%, 11: RobWzg=, 12:32, 13: Base=, 14:0, 15: SPSTrig=, 16:5, 17:[1/100s], 18: P, 19:19, 20:-1, 21:19
      ;FOLD 1: FB PSPS = EIN ;%{SE}%MKUKATPVW %CVW_SPS %VFBPSPS %P 2:FB PSPS = EIN,3:FBPSPS
      ;ENDFOLD
      ;FOLD 2: SPSMAKRO421 = EIN ;%{SE}%MKUKATPVW %CVW_SPS %VMAKRO %P 2:SPSMAKRO421 = EIN,3:MAKRO
      ;ENDFOLD
      ;FOLD 3: A23 = AUS ;%{SE}%MKUKATPVW %CVW_SPS %VBOASG %P 2:A23 = AUS,3:BOASG
      ;ENDFOLD
      ;FOLD 4: SPSMAKRO430 = EIN ;%{SE}%MKUKATPVW %CVW_SPS %VMAKRO %P 2:SPSMAKRO430 = EIN,3:MAKRO
      ;ENDFOLD
      ;FOLD 5: -- Werkzeug Kontrolle -- ;%{SE}%MKUKATPVW %CVW_COM %VCOMMENT %P 2:-- Werkzeug Kontrolle --,3:VW_COMMENT
      ;ENDFOLD
      ;FOLD 6: WARTE BIS E23 & M77 ;%{SE}%MKUKATPVW %CVW_SPS %VWBOASG %P 2:WARTE BIS E23 & M77,3:WBOASG
      ;ENDFOLD
      ;FOLD 7: A23 = EIN ;%{SE}%MKUKATPVW %CVW_SPS %VBOASG %P 2:A23 = EIN,3:BOASG
      ;ENDFOLD
      ;FOLD 8: FB PSPS = M30 & M77 & M81 & E548 & E549 & E551 ;%{SE}%MKUKATPVW %CVW_SPS %VFBPSPS %P 2:FB PSPS = M30 & M77 & M81 & E548 & E549 & E551,3:FBPSPS
      ;ENDFOLD
      ;FOLD {H}
         VW_MPARA_ACT=P19_D
         Act_P1 = P19
         Act_P2 = P19
         VW(#MPARA,TRUE)
         SPS_FERTIG=FALSE
         TRIGGER WHEN DISTANCE=1 DELAY=-50 DO SPS_TRIG(19) PRIO=-1
         LIN P19
         $ADVANCE=1
         WAIT FOR SPS_FERTIG
      ;ENDFOLD
   ;ENDFOLD
   ;FOLD -- Ueber  DB2 -- ;%{PSE}%MKUKATPVW,%CVW_COM,%VCOMMENT,%P 1:Comment:, 2:Ueber  DB2
      ;FOLD {H}
         M_COMMENT("Ueber  DB2")
      ;ENDFOLD
   ;ENDFOLD
   ;FOLD -- Profinet - Teilnehmer "Einschalten" -- ;%{PSE}%MKUKATPVW,%CVW_COM,%VCOMMENT,%P 1:Comment:, 2:Profinet - Teilnehmer "Einschalten"
      ;FOLD {H}
         M_COMMENT("Profinet - Teilnehmer Einschalten")
      ;ENDFOLD
   ;ENDFOLD
   ;FOLD LIN VB=50[mm/s] VE=0% ACC=100% RobWzg=32 Base=0 SPSTrig=5[1/100s] P ;%{P}%MKUKATPVW,%CMOVE8,%VLIN,%P 1:2, 2: VB=, 3:50, 4:[mm/s], 5: VE=, 6:0, 7:%, 8: ACC=, 9:100, 10:%, 11: RobWzg=, 12:32, 13: Base=, 14:0, 15: SPSTrig=, 16:5, 17:[1/100s], 18: P, 19:20, 20:-1, 21:20
      ;FOLD 1: FB PSPS = EIN ;%{SE}%MKUKATPVW %CVW_SPS %VFBPSPS %P 2:FB PSPS = EIN,3:FBPSPS
      ;ENDFOLD
      ;FOLD 2: A23 = AUS ;%{SE}%MKUKATPVW %CVW_SPS %VBOASG %P 2:A23 = AUS,3:BOASG
      ;ENDFOLD
      ;FOLD 3: WARTE BIS !E552 ;%{SE}%MKUKATPVW %CVW_SPS %VWBOASG %P 2:WARTE BIS !E552,3:WBOASG
      ;ENDFOLD
      ;FOLD 4: TECH3_ PN-Docken ID-Nr =122 Zuschalten EIN ;%{SE}%MKUKATPVW %CVW_SPS %VUSER %P 2:TECH3_.PN-Docken P1= 122 P2= 50 P3= 1 P4= 1 P5= 1 P6= 1 P7=EIN P8=301,3:USER
      ;ENDFOLD
      ;FOLD 5: WARTE ( EIN ) ZEIT 1 [1/10Sek] ;%{SE}%MKUKATPVW %CVW_SPS %VWTASG %P 2:WARTE ( EIN ) ZEIT 1 [1/10Sek],3:WTASG
      ;ENDFOLD
      ;FOLD 6: WARTE BIS E579 + E580 + E581 + E582 ;%{SE}%MKUKATPVW %CVW_SPS %VWBOASG %P 2:WARTE BIS E579 + E580 + E581 + E582,3:WBOASG
      ;ENDFOLD
      ;FOLD 7: -- Greifer Initialisieren -- ;%{SE}%MKUKATPVW %CVW_COM %VCOMMENT %P 2:-- Greifer Initialisieren --,3:VW_COMMENT
      ;ENDFOLD
      ;FOLD 8: F1 = EIN ;%{SE}%MKUKATPVW %CVW_SPS %VBOASG %P 2:F1 = EIN,3:BOASG
      ;ENDFOLD
      ;FOLD 9: SPSMAKRO343 = EIN ;%{SE}%MKUKATPVW %CVW_SPS %VMAKRO %P 2:SPSMAKRO343 = EIN,3:MAKRO
      ;ENDFOLD
      ;FOLD 10: F2 = EIN ;%{SE}%MKUKATPVW %CVW_SPS %VBOASG %P 2:F2 = EIN,3:BOASG
      ;ENDFOLD
      ;FOLD 11: SPSMAKRO342 = EIN ;%{SE}%MKUKATPVW %CVW_SPS %VMAKRO %P 2:SPSMAKRO342 = EIN,3:MAKRO
      ;ENDFOLD
      ;FOLD 12: SPSMAKRO340 = EIN ;%{SE}%MKUKATPVW %CVW_SPS %VMAKRO %P 2:SPSMAKRO340 = EIN,3:MAKRO
      ;ENDFOLD
      ;FOLD 13: WARTE BIS M32 & M33 ;%{SE}%MKUKATPVW %CVW_SPS %VWBOASG %P 2:WARTE BIS M32 & M33,3:WBOASG
      ;ENDFOLD
      ;FOLD 14: WARTE BIS E23 ;%{SE}%MKUKATPVW %CVW_SPS %VWBOASG %P 2:WARTE BIS E23,3:WBOASG
      ;ENDFOLD
      ;FOLD 15: A23 = EIN ;%{SE}%MKUKATPVW %CVW_SPS %VBOASG %P 2:A23 = EIN,3:BOASG
      ;ENDFOLD
      ;FOLD 16: FB PSPS = M30 & M32 & M33 & M77 & M83 & E548 & E549 ;%{SE}%MKUKATPVW %CVW_SPS %VFBPSPS %P 2:FB PSPS = M30 & M32 & M33 & M77 & M83 & E548 & E549,3:FBPSPS
      ;ENDFOLD
      ;FOLD {H}
         VW_MPARA_ACT=P20_D
         Act_P1 = P20
         Act_P2 = P20
         VW(#MPARA,TRUE)
         SPS_FERTIG=FALSE
         TRIGGER WHEN DISTANCE=1 DELAY=-50 DO SPS_TRIG(20) PRIO=-1
         VW_USER (#USR_ADV,301,122,50,1,1,1,1,TRUE)
         VW_USR_R (#USR_ADV,301,122,50,1,1,1,1,TRUE)
         LIN P20
         $ADVANCE=1
         WAIT FOR SPS_FERTIG
         VW_USER (#USR_MAIN,301,122,50,1,1,1,1,TRUE)
         VW_USR_R (#USR_MAIN,301,122,50,1,1,1,1,TRUE)
      ;ENDFOLD
   ;ENDFOLD
   ;FOLD LIN VB=200[mm/s] VE=10% ACC=100% RobWzg=32 Base=0 SPSTrig=0[1/100s] P ;%{P}%MKUKATPVW,%CMOVE8,%VLIN,%P 1:2, 2: VB=, 3:200, 4:[mm/s], 5: VE=, 6:10, 7:%, 8: ACC=, 9:100, 10:%, 11: RobWzg=, 12:32, 13: Base=, 14:0, 15: SPSTrig=, 16:0, 17:[1/100s], 18: P, 19:21, 20:-1, 21:21
      ;FOLD 1: FB PSPS = M30 & M32 & M33 & M77 & M83 & E548 & E549 ;%{SE}%MKUKATPVW %CVW_SPS %VFBPSPS %P 2:FB PSPS = M30 & M32 & M33 & M77 & M83 & E548 & E549,3:FBPSPS
      ;ENDFOLD
      ;FOLD {H}
         VW_MPARA_ACT=P21_D
         Act_P1 = P21
         Act_P2 = P21
         VW(#MPARA,TRUE)
         SPS_FERTIG=FALSE
         TRIGGER WHEN DISTANCE=1 DELAY=0 DO SPS_TRIG(10021) PRIO=-1
         LIN P21 C_VEL
         $ADVANCE=1
      ;ENDFOLD
   ;ENDFOLD
   ;FOLD LIN VB=800[mm/s] VE=100% ACC=100% RobWzg=32 Base=0 SPSTrig=0[1/100s] P ;%{P}%MKUKATPVW,%CMOVE8,%VLIN,%P 1:2, 2: VB=, 3:800, 4:[mm/s], 5: VE=, 6:100, 7:%, 8: ACC=, 9:100, 10:%, 11: RobWzg=, 12:32, 13: Base=, 14:0, 15: SPSTrig=, 16:0, 17:[1/100s], 18: P, 19:22, 20:-1, 21:22
      ;FOLD 1: FB PSPS = M30 & M32 & M33 & M77 & M83 & E548 & E549 ;%{SE}%MKUKATPVW %CVW_SPS %VFBPSPS %P 2:FB PSPS = M30 & M32 & M33 & M77 & M83 & E548 & E549,3:FBPSPS
      ;ENDFOLD
      ;FOLD {H}
         VW_MPARA_ACT=P22_D
         Act_P1 = P22
         Act_P2 = P22
         VW(#MPARA,TRUE)
         SPS_FERTIG=FALSE
         TRIGGER WHEN DISTANCE=1 DELAY=0 DO SPS_TRIG(10022) PRIO=-1
         LIN P22 C_VEL
         $ADVANCE=1
      ;ENDFOLD
   ;ENDFOLD
   ;FOLD PTP VB=100% VE=100% ACC=100% RobWzg=32 Base=0 SPSTrig=0[1/100s] P ;%{P}%MKUKATPVW,%CMOVE8,%VPTP,%P 1:1, 2: VB=, 3:100, 4:%, 5: VE=, 6:100, 7:%, 8: ACC=, 9:100, 10:%, 11: RobWzg=, 12:32, 13: Base=, 14:0, 15: SPSTrig=, 16:0, 17:[1/100s], 18: P, 19:23, 20:-1, 21:23
      ;FOLD 1: FB PSPS = M30 & M32 & M33 & M77 & M83 & E548 & E549 ;%{SE}%MKUKATPVW %CVW_SPS %VFBPSPS %P 2:FB PSPS = M30 & M32 & M33 & M77 & M83 & E548 & E549,3:FBPSPS
      ;ENDFOLD
      ;FOLD {H}
         VW_MPARA_ACT=P23_D
         Act_P1 = P23
         Act_P2 = P23
         VW(#MPARA,TRUE)
         SPS_FERTIG=FALSE
         TRIGGER WHEN DISTANCE=1 DELAY=0 DO SPS_TRIG(10023) PRIO=-1
         PTP P23 C_PTP C_VEL
         $ADVANCE=1
      ;ENDFOLD
   ;ENDFOLD
   ;FOLD PTP VB=100% VE=100% ACC=100% RobWzg=32 Base=0 SPSTrig=0[1/100s] P ;%{P}%MKUKATPVW,%CMOVE8,%VPTP,%P 1:1, 2: VB=, 3:100, 4:%, 5: VE=, 6:100, 7:%, 8: ACC=, 9:100, 10:%, 11: RobWzg=, 12:32, 13: Base=, 14:0, 15: SPSTrig=, 16:0, 17:[1/100s], 18: P, 19:24, 20:-1, 21:24
      ;FOLD 1: FB PSPS = M30 & M32 & M33 & M77 & M83 & E548 & E549 ;%{SE}%MKUKATPVW %CVW_SPS %VFBPSPS %P 2:FB PSPS = M30 & M32 & M33 & M77 & M83 & E548 & E549,3:FBPSPS
      ;ENDFOLD
      ;FOLD {H}
         VW_MPARA_ACT=P24_D
         Act_P1 = P24
         Act_P2 = P24
         VW(#MPARA,TRUE)
         SPS_FERTIG=FALSE
         TRIGGER WHEN DISTANCE=1 DELAY=0 DO SPS_TRIG(10024) PRIO=-1
         PTP P24 C_PTP C_VEL
         $ADVANCE=1
      ;ENDFOLD
   ;ENDFOLD
   ;FOLD PTP VB=100% VE=100% ACC=100% RobWzg=32 Base=0 SPSTrig=0[1/100s] P ;%{P}%MKUKATPVW,%CMOVE8,%VPTP,%P 1:1, 2: VB=, 3:100, 4:%, 5: VE=, 6:100, 7:%, 8: ACC=, 9:100, 10:%, 11: RobWzg=, 12:32, 13: Base=, 14:0, 15: SPSTrig=, 16:0, 17:[1/100s], 18: P, 19:25, 20:-1, 21:25
      ;FOLD 1: FB PSPS = M30 & M32 & M33 & M77 & M83 & E548 & E549 ;%{SE}%MKUKATPVW %CVW_SPS %VFBPSPS %P 2:FB PSPS = M30 & M32 & M33 & M77 & M83 & E548 & E549,3:FBPSPS
      ;ENDFOLD
      ;FOLD {H}
         VW_MPARA_ACT=P25_D
         Act_P1 = P25
         Act_P2 = P25
         VW(#MPARA,TRUE)
         SPS_FERTIG=FALSE
         TRIGGER WHEN DISTANCE=1 DELAY=0 DO SPS_TRIG(10025) PRIO=-1
         PTP P25 C_PTP C_VEL
         $ADVANCE=1
      ;ENDFOLD
   ;ENDFOLD
   ;FOLD -- DB2 Abdeckklappe ZU -- ;%{PSE}%MKUKATPVW,%CVW_COM,%VCOMMENT,%P 1:Comment:, 2:DB2 Abdeckklappe ZU
      ;FOLD {H}
         M_COMMENT("DB2 Abdeckklappe ZU")
      ;ENDFOLD
   ;ENDFOLD
   ;FOLD PTP VB=100% VE=0% ACC=100% RobWzg=32 Base=0 SPSTrig=0[1/100s] P ;%{P}%MKUKATPVW,%CMOVE8,%VPTP,%P 1:1, 2: VB=, 3:100, 4:%, 5: VE=, 6:0, 7:%, 8: ACC=, 9:100, 10:%, 11: RobWzg=, 12:32, 13: Base=, 14:0, 15: SPSTrig=, 16:0, 17:[1/100s], 18: P, 19:26, 20:-1, 21:26
      ;FOLD 1: FB PSPS = EIN ;%{SE}%MKUKATPVW %CVW_SPS %VFBPSPS %P 2:FB PSPS = EIN,3:FBPSPS
      ;ENDFOLD
      ;FOLD 2: A23 = AUS ;%{SE}%MKUKATPVW %CVW_SPS %VBOASG %P 2:A23 = AUS,3:BOASG
      ;ENDFOLD
      ;FOLD 3: SPSMAKRO430 = EIN ;%{SE}%MKUKATPVW %CVW_SPS %VMAKRO %P 2:SPSMAKRO430 = EIN,3:MAKRO
      ;ENDFOLD
      ;FOLD 4: F841 = EIN ;%{SE}%MKUKATPVW %CVW_SPS %VBOASG %P 2:F841 = EIN,3:BOASG
      ;ENDFOLD
      ;FOLD 5: F842 = EIN ;%{SE}%MKUKATPVW %CVW_SPS %VBOASG %P 2:F842 = EIN,3:BOASG
      ;ENDFOLD
      ;FOLD 6: SPSMAKRO433 = EIN ;%{SE}%MKUKATPVW %CVW_SPS %VMAKRO %P 2:SPSMAKRO433 = EIN,3:MAKRO
      ;ENDFOLD
      ;FOLD 7: WARTE BIS !E547 & E548 & !E549 & E550 ;%{SE}%MKUKATPVW %CVW_SPS %VWBOASG %P 2:WARTE BIS !E547 & E548 & !E549 & E550,3:WBOASG
      ;ENDFOLD
      ;FOLD 8: SPSMAKRO430 = EIN ;%{SE}%MKUKATPVW %CVW_SPS %VMAKRO %P 2:SPSMAKRO430 = EIN,3:MAKRO
      ;ENDFOLD
      ;FOLD 9: t6 ( EIN ) = STOP ;%{SE}%MKUKATPVW %CVW_SPS %VTSTOP %P 2:t6 ( EIN ) = STOP,3:TSTOP
      ;ENDFOLD
      ;FOLD 10: WARTE BIS E23 ;%{SE}%MKUKATPVW %CVW_SPS %VWBOASG %P 2:WARTE BIS E23,3:WBOASG
      ;ENDFOLD
      ;FOLD 11: A23 = EIN ;%{SE}%MKUKATPVW %CVW_SPS %VBOASG %P 2:A23 = EIN,3:BOASG
      ;ENDFOLD
      ;FOLD 12: FB PSPS = M13 & M30 & M32 & M33 & M77 ;%{SE}%MKUKATPVW %CVW_SPS %VFBPSPS %P 2:FB PSPS = M13 & M30 & M32 & M33 & M77,3:FBPSPS
      ;ENDFOLD
      ;FOLD {H}
         VW_MPARA_ACT=P26_D
         Act_P1 = P26
         Act_P2 = P26
         VW(#MPARA,TRUE)
         SPS_FERTIG=FALSE
         TRIGGER WHEN DISTANCE=1 DELAY=0 DO SPS_TRIG(26) PRIO=-1
         PTP P26
         $ADVANCE=1
         WAIT FOR SPS_FERTIG
      ;ENDFOLD
   ;ENDFOLD
   ; FOLD ;%{H}
END
DEF SPS_TRIG(NO :IN)
   INT NO
   INT VW_STOP
   BOOL UES
   VW_STOP=$VW_PSPS_STOP
   IF NO>10000 THEN
      NO=NO-10000
      UES=TRUE
   ELSE
      UES=FALSE
   ENDIF
   ; FOLD ;%{H}
   IF ((VW_STOP B_AND 'B0001') > 0) THEN
      ;-- Trigger vorzeitig geschaltet (delay < 0) oder MStep
      IF (((VW_STOP B_AND 'B0110') > 0) AND ($MODE_OP<>#EX)) THEN
         ;-- MStep oder BCO Bewegung
         HALT
      ENDIF
   ENDIF
   ; ENDFOLD
   IF (SEARCH_END) THEN
      SEARCH_END = FALSE
      INTERRUPT OFF 39
   ENDIF
   SWITCH NO
      CASE 1
         ;FOLD SPS_TRIG1{H}
            VALCYCFL30=$CYCFLAG[254]
            $CYCFLAG[254]=(FALSE) AND $CYCFLAG[255] OR ($TIMER[61]<0)
            VW(#FB_CHECK,TRUE)
            $OUT[23] = FALSE
            VW(#SET_TIME,TRUE,6,0,0)
            SEL_RES=SELECT(#MAKRO,50,TRUE,,,,,FALSE)
            SEL_RES=SELECT(#MAKRO,53,TRUE,,,,,FALSE)
            $OUT[42] = TRUE
            $OUT[43] = TRUE
            $OUT[44] = TRUE
            $OUT[45] = TRUE
            $OUT[47] = TRUE
            $OUT[49] = TRUE
            $OUT[52] = TRUE
            $OUT[54] = TRUE
            $OUT[75] = TRUE
            $OUT[76] = TRUE
            $OUT[79] = TRUE
            $OUT[80] = TRUE
            $LOOP_MSG[]="M13 & M78 & !E16"
            $LOOP_CONT=TRUE
            WAIT FOR ($CYCFLAG[13] AND $CYCFLAG[78] AND NOT $IN[16]) OR (NOT $LOOP_CONT AND ($MODE_OP<>#EX))
            $LOOP_MSG[]="                                                                                                                                "
            $FLAG[1] = TRUE
            $FLAG[2] = TRUE
            SEL_RES=SELECT(#MAKRO,343,$CYCFLAG[13],,,,,FALSE)
            SEL_RES=SELECT(#MAKRO,340,TRUE,,,,,FALSE)
            $LOOP_MSG[]="M32 & M34"
            $LOOP_CONT=TRUE
            WAIT FOR ($CYCFLAG[32] AND $CYCFLAG[34]) OR (NOT $LOOP_CONT AND ($MODE_OP<>#EX))
            $LOOP_MSG[]="                                                                                                                                "
            SEL_RES=SELECT(#MAKRO,430,TRUE,,,,,FALSE)
            $FLAG[841] = TRUE
            $FLAG[842] = TRUE
            SEL_RES=SELECT(#MAKRO,432,TRUE,,,,,FALSE)
            $LOOP_MSG[]="E547 & !E548 & E549 & !E550 & E552"
            $LOOP_CONT=TRUE
            WAIT FOR ($IN[547] AND NOT $IN[548] AND $IN[549] AND NOT $IN[550] AND $IN[552]) OR (NOT $LOOP_CONT AND ($MODE_OP<>#EX))
            $LOOP_MSG[]="                                                                                                                                "
            $LOOP_MSG[]="E23"
            $LOOP_CONT=TRUE
            WAIT FOR ($IN[23]) OR (NOT $LOOP_CONT AND ($MODE_OP<>#EX))
            $LOOP_MSG[]="                                                                                                                                "
            $OUT[23] = TRUE
            VALCYCFL30=$CYCFLAG[254]
            $CYCFLAG[254]=($CYCFLAG[30] AND $CYCFLAG[32] AND $CYCFLAG[34] AND $CYCFLAG[78] AND $CYCFLAG[82] AND $IN[547] AND $IN[549]) AND $CYCFLAG[255] OR ($TIMER[61]<0)
            VW(#FB_CHECK,TRUE)
         ;ENDFOLD
      CASE 2
         ;FOLD SPS_TRIG2{H}
            VALCYCFL30=$CYCFLAG[254]
            $CYCFLAG[254]=($CYCFLAG[30] AND $CYCFLAG[32] AND $CYCFLAG[34] AND $CYCFLAG[78] AND $CYCFLAG[82] AND $IN[547] AND $IN[549]) AND $CYCFLAG[255] OR ($TIMER[61]<0)
            VW(#FB_CHECK,TRUE)
         ;ENDFOLD
      CASE 3
         ;FOLD SPS_TRIG3{H}
            VALCYCFL30=$CYCFLAG[254]
            $CYCFLAG[254]=($CYCFLAG[30] AND $CYCFLAG[32] AND $CYCFLAG[34] AND $CYCFLAG[78] AND $CYCFLAG[82] AND $IN[547] AND $IN[549]) AND $CYCFLAG[255] OR ($TIMER[61]<0)
            VW(#FB_CHECK,TRUE)
         ;ENDFOLD
      CASE 4
         ;FOLD SPS_TRIG4{H}
            VALCYCFL30=$CYCFLAG[254]
            $CYCFLAG[254]=($CYCFLAG[30] AND $CYCFLAG[32] AND $CYCFLAG[34] AND $CYCFLAG[78] AND $CYCFLAG[82] AND $IN[547] AND $IN[549]) AND $CYCFLAG[255] OR ($TIMER[61]<0)
            VW(#FB_CHECK,TRUE)
         ;ENDFOLD
      CASE 5
         ;FOLD SPS_TRIG5{H}
            VALCYCFL30=$CYCFLAG[254]
            $CYCFLAG[254]=($CYCFLAG[30] AND $CYCFLAG[32] AND $CYCFLAG[34] AND $CYCFLAG[78] AND $CYCFLAG[82] AND $IN[547] AND $IN[549]) AND $CYCFLAG[255] OR ($TIMER[61]<0)
            VW(#FB_CHECK,TRUE)
         ;ENDFOLD
      CASE 6
         ;FOLD SPS_TRIG6{H}
            VALCYCFL30=$CYCFLAG[254]
            $CYCFLAG[254]=(TRUE) AND $CYCFLAG[255] OR ($TIMER[61]<0)
            VW(#FB_CHECK,TRUE)
            $OUT[23] = FALSE
            SEL_RES=SELECT(#MAKRO,422,NOT $IN[540],,,,,FALSE)
            $LOOP_MSG[]="E540 & !E551 & E23"
            $LOOP_CONT=TRUE
            WAIT FOR ($IN[540] AND NOT $IN[551] AND $IN[23]) OR (NOT $LOOP_CONT AND ($MODE_OP<>#EX))
            $LOOP_MSG[]="                                                                                                                                "
            VW_USER (#USR_TRIG,301,122,60,1,1,1,1,TRUE)
            VW_USR_R (#USR_TRIG,301,122,60,1,1,1,1,TRUE)
            $OUT[23] = TRUE
            VALCYCFL30=$CYCFLAG[254]
            $CYCFLAG[254]=($CYCFLAG[30] AND $CYCFLAG[78] AND $IN[547] AND $IN[549]) AND $CYCFLAG[255] OR ($TIMER[61]<0)
            VW(#FB_CHECK,TRUE)
         ;ENDFOLD
      CASE 7
         ;FOLD SPS_TRIG7{H}
            VALCYCFL30=$CYCFLAG[254]
            $CYCFLAG[254]=($CYCFLAG[30] AND $CYCFLAG[78] AND $IN[547] AND $IN[549]) AND $CYCFLAG[255] OR ($TIMER[61]<0)
            VW(#FB_CHECK,TRUE)
         ;ENDFOLD
      CASE 8
         ;FOLD SPS_TRIG8{H}
            VALCYCFL30=$CYCFLAG[254]
            $CYCFLAG[254]=(TRUE) AND $CYCFLAG[255] OR ($TIMER[61]<0)
            VW(#FB_CHECK,TRUE)
            $OUT[23] = FALSE
            $LOOP_MSG[]="E540 & E551 & E23"
            $LOOP_CONT=TRUE
            WAIT FOR ($IN[540] AND $IN[551] AND $IN[23]) OR (NOT $LOOP_CONT AND ($MODE_OP<>#EX))
            $LOOP_MSG[]="                                                                                                                                "
            $OUT[23] = TRUE
            SEL_RES=SELECT(#MAKRO,420,TRUE,,,,,FALSE)
            $LOOP_MSG[]="!E538 & E539"
            $LOOP_CONT=TRUE
            WAIT FOR (NOT $IN[538] AND $IN[539]) OR (NOT $LOOP_CONT AND ($MODE_OP<>#EX))
            $LOOP_MSG[]="                                                                                                                                "
            VALCYCFL30=$CYCFLAG[254]
            $CYCFLAG[254]=($CYCFLAG[30] AND NOT $IN[538] AND $IN[539] AND $IN[540] AND $IN[551] AND $IN[552]) AND $CYCFLAG[255] OR ($TIMER[61]<0)
            VW(#FB_CHECK,TRUE)
         ;ENDFOLD
      CASE 9
         ;FOLD SPS_TRIG9{H}
            VALCYCFL30=$CYCFLAG[254]
            $CYCFLAG[254]=($CYCFLAG[30] AND $IN[547] AND $IN[549] AND $IN[551] AND $IN[552]) AND $CYCFLAG[255] OR ($TIMER[61]<0)
            VW(#FB_CHECK,TRUE)
         ;ENDFOLD
      CASE 10
         ;FOLD SPS_TRIG10{H}
            VALCYCFL30=$CYCFLAG[254]
            $CYCFLAG[254]=(TRUE) AND $CYCFLAG[255] OR ($TIMER[61]<0)
            VW(#FB_CHECK,TRUE)
            $OUT[539] = FALSE
            VALCYCFL30=$CYCFLAG[254]
            $CYCFLAG[254]=($CYCFLAG[30] AND $IN[547] AND $IN[549] AND $IN[551] AND $IN[552]) AND $CYCFLAG[255] OR ($TIMER[61]<0)
            VW(#FB_CHECK,TRUE)
         ;ENDFOLD
      CASE 11
         ;FOLD SPS_TRIG11{H}
            VALCYCFL30=$CYCFLAG[254]
            $CYCFLAG[254]=($CYCFLAG[30] AND $IN[547] AND $IN[549] AND $IN[551] AND $IN[552]) AND $CYCFLAG[255] OR ($TIMER[61]<0)
            VW(#FB_CHECK,TRUE)
         ;ENDFOLD
      CASE 12
         ;FOLD SPS_TRIG12{H}
            VALCYCFL30=$CYCFLAG[254]
            $CYCFLAG[254]=($CYCFLAG[30] AND $IN[547] AND $IN[549] AND $IN[551] AND $IN[552]) AND $CYCFLAG[255] OR ($TIMER[61]<0)
            VW(#FB_CHECK,TRUE)
         ;ENDFOLD
      CASE 13
         ;FOLD SPS_TRIG13{H}
            VALCYCFL30=$CYCFLAG[254]
            $CYCFLAG[254]=(TRUE) AND $CYCFLAG[255] OR ($TIMER[61]<0)
            VW(#FB_CHECK,TRUE)
            $FLAG[842] = TRUE
            SEL_RES=SELECT(#MAKRO,433,TRUE,,,,,FALSE)
            $FLAG[841] = TRUE
            SEL_RES=SELECT(#MAKRO,432,TRUE,,,,,FALSE)
            $LOOP_MSG[]="E549 & !E550 & E23"
            $LOOP_CONT=TRUE
            WAIT FOR ($IN[549] AND NOT $IN[550] AND $IN[23]) OR (NOT $LOOP_CONT AND ($MODE_OP<>#EX))
            $LOOP_MSG[]="                                                                                                                                "
            $OUT[539] = FALSE
            $OUT[23] = FALSE
            $LOOP_MSG[]="E23"
            $LOOP_CONT=TRUE
            WAIT FOR ($IN[23]) OR (NOT $LOOP_CONT AND ($MODE_OP<>#EX))
            $LOOP_MSG[]="                                                                                                                                "
            $OUT[23] = TRUE
            $FLAG[958] = NOT $FLAG[933]
            VALCYCFL30=$CYCFLAG[254]
            $CYCFLAG[254]=($CYCFLAG[30] AND NOT $IN[547] AND $IN[548] AND $IN[549] AND $IN[551] AND $IN[552]) AND $CYCFLAG[255] OR ($TIMER[61]<0)
            VW(#FB_CHECK,TRUE)
         ;ENDFOLD
      CASE 14
         ;FOLD SPS_TRIG14{H}
            VALCYCFL30=$CYCFLAG[254]
            $CYCFLAG[254]=(TRUE) AND $CYCFLAG[255] OR ($TIMER[61]<0)
            VW(#FB_CHECK,TRUE)
            $OUT[23] = FALSE
            $FLAG[841] = TRUE
            $FLAG[842] = TRUE
            SEL_RES=SELECT(#MAKRO,433,TRUE,,,,,FALSE)
            $LOOP_MSG[]="!E549 & E550 & !E547 & E548 & E23"
            $LOOP_CONT=TRUE
            WAIT FOR (NOT $IN[549] AND $IN[550] AND NOT $IN[547] AND $IN[548] AND $IN[23]) OR (NOT $LOOP_CONT AND ($MODE_OP<>#EX))
            $LOOP_MSG[]="                                                                                                                                "
            SEL_RES=SELECT(#MAKRO,430,TRUE,,,,,FALSE)
            $OUT[17] = TRUE
            VW(#BINOUT,TRUE,19,0)
            $LOOP_MSG[]="E17"
            $LOOP_CONT=TRUE
            WAIT FOR ($IN[17]) OR (NOT $LOOP_CONT AND ($MODE_OP<>#EX))
            $LOOP_MSG[]="                                                                                                                                "
            $OUT[17] = FALSE
            $FLAG[933] = FALSE
            $FLAG[958] = FALSE
            $FLAG[841] = TRUE
            SEL_RES=SELECT(#MAKRO,432,TRUE,,,,,FALSE)
            $LOOP_MSG[]="E549 & !E550"
            $LOOP_CONT=TRUE
            WAIT FOR ($IN[549] AND NOT $IN[550]) OR (NOT $LOOP_CONT AND ($MODE_OP<>#EX))
            $LOOP_MSG[]="                                                                                                                                "
            $LOOP_MSG[]="E23"
            $LOOP_CONT=TRUE
            WAIT FOR ($IN[23]) OR (NOT $LOOP_CONT AND ($MODE_OP<>#EX))
            $LOOP_MSG[]="                                                                                                                                "
            $OUT[23] = TRUE
            VALCYCFL30=$CYCFLAG[254]
            $CYCFLAG[254]=($CYCFLAG[30] AND NOT $IN[547] AND $IN[548] AND $IN[549] AND $IN[551] AND $IN[552]) AND $CYCFLAG[255] OR ($TIMER[61]<0)
            VW(#FB_CHECK,TRUE)
         ;ENDFOLD
      CASE 15
         ;FOLD SPS_TRIG15{H}
            VALCYCFL30=$CYCFLAG[254]
            $CYCFLAG[254]=(TRUE) AND $CYCFLAG[255] OR ($TIMER[61]<0)
            VW(#FB_CHECK,TRUE)
            $OUT[23] = FALSE
            SEL_RES=SELECT(#MAKRO,422,NOT $IN[540],,,,,FALSE)
            $LOOP_MSG[]="E540 & E23"
            $LOOP_CONT=TRUE
            WAIT FOR ($IN[540] AND $IN[23]) OR (NOT $LOOP_CONT AND ($MODE_OP<>#EX))
            $LOOP_MSG[]="                                                                                                                                "
            $OUT[23] = TRUE
            VALCYCFL30=$CYCFLAG[254]
            $CYCFLAG[254]=($CYCFLAG[30] AND NOT $IN[547] AND $IN[548] AND $IN[549] AND $IN[551] AND $IN[552]) AND $CYCFLAG[255] OR ($TIMER[61]<0)
            VW(#FB_CHECK,TRUE)
         ;ENDFOLD
      CASE 16
         ;FOLD SPS_TRIG16{H}
            VALCYCFL30=$CYCFLAG[254]
            $CYCFLAG[254]=($CYCFLAG[30] AND NOT $IN[547] AND $IN[548] AND $IN[549] AND $IN[551] AND $IN[552]) AND $CYCFLAG[255] OR ($TIMER[61]<0)
            VW(#FB_CHECK,TRUE)
         ;ENDFOLD
      CASE 17
         ;FOLD SPS_TRIG17{H}
            VALCYCFL30=$CYCFLAG[254]
            $CYCFLAG[254]=($CYCFLAG[30] AND NOT $IN[547] AND $IN[548] AND $IN[549] AND $IN[551] AND $IN[552]) AND $CYCFLAG[255] OR ($TIMER[61]<0)
            VW(#FB_CHECK,TRUE)
         ;ENDFOLD
      CASE 18
         ;FOLD SPS_TRIG18{H}
            VALCYCFL30=$CYCFLAG[254]
            $CYCFLAG[254]=(TRUE) AND $CYCFLAG[255] OR ($TIMER[61]<0)
            VW(#FB_CHECK,TRUE)
            $OUT[23] = FALSE
            $LOOP_MSG[]="E23"
            $LOOP_CONT=TRUE
            WAIT FOR ($IN[23]) OR (NOT $LOOP_CONT AND ($MODE_OP<>#EX))
            $LOOP_MSG[]="                                                                                                                                "
            $OUT[23] = TRUE
            SEL_RES=SELECT(#MAKRO,52,TRUE,,,,,FALSE)
            $OUT[539] = TRUE
            $LOOP_MSG[]="!E538 & E539 & E540"
            $LOOP_CONT=TRUE
            WAIT FOR (NOT $IN[538] AND $IN[539] AND $IN[540]) OR (NOT $LOOP_CONT AND ($MODE_OP<>#EX))
            $LOOP_MSG[]="                                                                                                                                "
            VALCYCFL30=$CYCFLAG[254]
            $CYCFLAG[254]=($CYCFLAG[30] AND NOT $IN[538] AND $IN[539] AND $IN[548] AND $IN[549] AND $IN[551] AND $IN[552]) AND $CYCFLAG[255] OR ($TIMER[61]<0)
            VW(#FB_CHECK,TRUE)
         ;ENDFOLD
      CASE 19
         ;FOLD SPS_TRIG19{H}
            VALCYCFL30=$CYCFLAG[254]
            $CYCFLAG[254]=(TRUE) AND $CYCFLAG[255] OR ($TIMER[61]<0)
            VW(#FB_CHECK,TRUE)
            SEL_RES=SELECT(#MAKRO,421,TRUE,,,,,FALSE)
            $OUT[23] = FALSE
            SEL_RES=SELECT(#MAKRO,430,TRUE,,,,,FALSE)
            $LOOP_MSG[]="E23 & M77"
            $LOOP_CONT=TRUE
            WAIT FOR ($IN[23] AND $CYCFLAG[77]) OR (NOT $LOOP_CONT AND ($MODE_OP<>#EX))
            $LOOP_MSG[]="                                                                                                                                "
            $OUT[23] = TRUE
            VALCYCFL30=$CYCFLAG[254]
            $CYCFLAG[254]=($CYCFLAG[30] AND $CYCFLAG[77] AND $CYCFLAG[81] AND $IN[548] AND $IN[549] AND $IN[551]) AND $CYCFLAG[255] OR ($TIMER[61]<0)
            VW(#FB_CHECK,TRUE)
         ;ENDFOLD
      CASE 20
         ;FOLD SPS_TRIG20{H}
            VALCYCFL30=$CYCFLAG[254]
            $CYCFLAG[254]=(TRUE) AND $CYCFLAG[255] OR ($TIMER[61]<0)
            VW(#FB_CHECK,TRUE)
            $OUT[23] = FALSE
            $LOOP_MSG[]="!E552"
            $LOOP_CONT=TRUE
            WAIT FOR (NOT $IN[552]) OR (NOT $LOOP_CONT AND ($MODE_OP<>#EX))
            $LOOP_MSG[]="                                                                                                                                "
            VW_USER (#USR_TRIG,301,122,50,1,1,1,1,TRUE)
            VW_USR_R (#USR_TRIG,301,122,50,1,1,1,1,TRUE)
            $LOOP_MSG[]="Wartezeit..."
            $LOOP_CONT=TRUE
            WAIT FOR (FALSE OR TIMER_LIMIT ((1)*0.1) OR (NOT $LOOP_CONT AND ($MODE_OP<>#EX)))
            $LOOP_MSG[]="                                                                                                                                "
            $LOOP_MSG[]="E579 + E580 + E581 + E582"
            $LOOP_CONT=TRUE
            WAIT FOR ($IN[579] OR $IN[580] OR $IN[581] OR $IN[582]) OR (NOT $LOOP_CONT AND ($MODE_OP<>#EX))
            $LOOP_MSG[]="                                                                                                                                "
            $FLAG[1] = TRUE
            SEL_RES=SELECT(#MAKRO,343,TRUE,,,,,FALSE)
            $FLAG[2] = TRUE
            SEL_RES=SELECT(#MAKRO,342,TRUE,,,,,FALSE)
            SEL_RES=SELECT(#MAKRO,340,TRUE,,,,,FALSE)
            $LOOP_MSG[]="M32 & M33"
            $LOOP_CONT=TRUE
            WAIT FOR ($CYCFLAG[32] AND $CYCFLAG[33]) OR (NOT $LOOP_CONT AND ($MODE_OP<>#EX))
            $LOOP_MSG[]="                                                                                                                                "
            $LOOP_MSG[]="E23"
            $LOOP_CONT=TRUE
            WAIT FOR ($IN[23]) OR (NOT $LOOP_CONT AND ($MODE_OP<>#EX))
            $LOOP_MSG[]="                                                                                                                                "
            $OUT[23] = TRUE
            VALCYCFL30=$CYCFLAG[254]
            $CYCFLAG[254]=($CYCFLAG[30] AND $CYCFLAG[32] AND $CYCFLAG[33] AND $CYCFLAG[77] AND $CYCFLAG[83] AND $IN[548] AND $IN[549]) AND $CYCFLAG[255] OR ($TIMER[61]<0)
            VW(#FB_CHECK,TRUE)
         ;ENDFOLD
      CASE 21
         ;FOLD SPS_TRIG21{H}
            VALCYCFL30=$CYCFLAG[254]
            $CYCFLAG[254]=($CYCFLAG[30] AND $CYCFLAG[32] AND $CYCFLAG[33] AND $CYCFLAG[77] AND $CYCFLAG[83] AND $IN[548] AND $IN[549]) AND $CYCFLAG[255] OR ($TIMER[61]<0)
            VW(#FB_CHECK,TRUE)
         ;ENDFOLD
      CASE 22
         ;FOLD SPS_TRIG22{H}
            VALCYCFL30=$CYCFLAG[254]
            $CYCFLAG[254]=($CYCFLAG[30] AND $CYCFLAG[32] AND $CYCFLAG[33] AND $CYCFLAG[77] AND $CYCFLAG[83] AND $IN[548] AND $IN[549]) AND $CYCFLAG[255] OR ($TIMER[61]<0)
            VW(#FB_CHECK,TRUE)
         ;ENDFOLD
      CASE 23
         ;FOLD SPS_TRIG23{H}
            VALCYCFL30=$CYCFLAG[254]
            $CYCFLAG[254]=($CYCFLAG[30] AND $CYCFLAG[32] AND $CYCFLAG[33] AND $CYCFLAG[77] AND $CYCFLAG[83] AND $IN[548] AND $IN[549]) AND $CYCFLAG[255] OR ($TIMER[61]<0)
            VW(#FB_CHECK,TRUE)
         ;ENDFOLD
      CASE 24
         ;FOLD SPS_TRIG24{H}
            VALCYCFL30=$CYCFLAG[254]
            $CYCFLAG[254]=($CYCFLAG[30] AND $CYCFLAG[32] AND $CYCFLAG[33] AND $CYCFLAG[77] AND $CYCFLAG[83] AND $IN[548] AND $IN[549]) AND $CYCFLAG[255] OR ($TIMER[61]<0)
            VW(#FB_CHECK,TRUE)
         ;ENDFOLD
      CASE 25
         ;FOLD SPS_TRIG25{H}
            VALCYCFL30=$CYCFLAG[254]
            $CYCFLAG[254]=($CYCFLAG[30] AND $CYCFLAG[32] AND $CYCFLAG[33] AND $CYCFLAG[77] AND $CYCFLAG[83] AND $IN[548] AND $IN[549]) AND $CYCFLAG[255] OR ($TIMER[61]<0)
            VW(#FB_CHECK,TRUE)
         ;ENDFOLD
      CASE 26
         ;FOLD SPS_TRIG26{H}
            VALCYCFL30=$CYCFLAG[254]
            $CYCFLAG[254]=(TRUE) AND $CYCFLAG[255] OR ($TIMER[61]<0)
            VW(#FB_CHECK,TRUE)
            $OUT[23] = FALSE
            SEL_RES=SELECT(#MAKRO,430,TRUE,,,,,FALSE)
            $FLAG[841] = TRUE
            $FLAG[842] = TRUE
            SEL_RES=SELECT(#MAKRO,433,TRUE,,,,,FALSE)
            $LOOP_MSG[]="!E547 & E548 & !E549 & E550"
            $LOOP_CONT=TRUE
            WAIT FOR (NOT $IN[547] AND $IN[548] AND NOT $IN[549] AND $IN[550]) OR (NOT $LOOP_CONT AND ($MODE_OP<>#EX))
            $LOOP_MSG[]="                                                                                                                                "
            SEL_RES=SELECT(#MAKRO,430,TRUE,,,,,FALSE)
            VW(#SET_TIME,TRUE,6,1,0)
            $LOOP_MSG[]="E23"
            $LOOP_CONT=TRUE
            WAIT FOR ($IN[23]) OR (NOT $LOOP_CONT AND ($MODE_OP<>#EX))
            $LOOP_MSG[]="                                                                                                                                "
            $OUT[23] = TRUE
            VALCYCFL30=$CYCFLAG[254]
            $CYCFLAG[254]=($CYCFLAG[13] AND $CYCFLAG[30] AND $CYCFLAG[32] AND $CYCFLAG[33] AND $CYCFLAG[77]) AND $CYCFLAG[255] OR ($TIMER[61]<0)
            VW(#FB_CHECK,TRUE)
         ;ENDFOLD
      CASE 27
         ;FOLD SPS_TRIG27{H}
         ;ENDFOLD
      CASE 28
         ;FOLD SPS_TRIG28{H}
         ;ENDFOLD
      CASE 29
         ;FOLD SPS_TRIG29{H}
         ;ENDFOLD
      CASE 30
         ;FOLD SPS_TRIG30{H}
         ;ENDFOLD
      CASE 31
         ;FOLD SPS_TRIG31{H}
         ;ENDFOLD
      CASE 32
         ;FOLD SPS_TRIG32{H}
         ;ENDFOLD
      CASE 33
         ;FOLD SPS_TRIG33{H}
         ;ENDFOLD
      CASE 34
         ;FOLD SPS_TRIG34{H}
         ;ENDFOLD
      CASE 35
         ;FOLD SPS_TRIG35{H}
         ;ENDFOLD
      CASE 36
         ;FOLD SPS_TRIG36{H}
         ;ENDFOLD
      CASE 37
         ;FOLD SPS_TRIG37{H}
         ;ENDFOLD
      CASE 38
         ;FOLD SPS_TRIG38{H}
         ;ENDFOLD
      CASE 39
         ;FOLD SPS_TRIG39{H}
         ;ENDFOLD
      CASE 40
         ;FOLD SPS_TRIG40{H}
         ;ENDFOLD
      CASE 41
         ;FOLD SPS_TRIG41{H}
         ;ENDFOLD
      CASE 42
         ;FOLD SPS_TRIG42{H}
         ;ENDFOLD
      CASE 43
         ;FOLD SPS_TRIG43{H}
         ;ENDFOLD
      CASE 44
         ;FOLD SPS_TRIG44{H}
         ;ENDFOLD
      CASE 45
         ;FOLD SPS_TRIG45{H}
         ;ENDFOLD
      CASE 46
         ;FOLD SPS_TRIG46{H}
         ;ENDFOLD
      CASE 47
         ;FOLD SPS_TRIG47{H}
         ;ENDFOLD
      CASE 48
         ;FOLD SPS_TRIG48{H}
         ;ENDFOLD
      CASE 49
         ;FOLD SPS_TRIG49{H}
         ;ENDFOLD
      CASE 50
         ;FOLD SPS_TRIG50{H}
         ;ENDFOLD
      CASE 51
         ;FOLD SPS_TRIG51{H}
         ;ENDFOLD
      CASE 52
         ;FOLD SPS_TRIG52{H}
         ;ENDFOLD
      CASE 53
         ;FOLD SPS_TRIG53{H}
         ;ENDFOLD
      CASE 54
         ;FOLD SPS_TRIG54{H}
         ;ENDFOLD
      CASE 55
         ;FOLD SPS_TRIG55{H}
         ;ENDFOLD
      CASE 56
         ;FOLD SPS_TRIG56{H}
         ;ENDFOLD
      CASE 57
         ;FOLD SPS_TRIG57{H}
         ;ENDFOLD
      CASE 58
         ;FOLD SPS_TRIG58{H}
         ;ENDFOLD
      CASE 59
         ;FOLD SPS_TRIG59{H}
         ;ENDFOLD
      CASE 60
         ;FOLD SPS_TRIG60{H}
         ;ENDFOLD
      CASE 61
         ;FOLD SPS_TRIG61{H}
         ;ENDFOLD
      CASE 62
         ;FOLD SPS_TRIG62{H}
         ;ENDFOLD
      CASE 63
         ;FOLD SPS_TRIG63{H}
         ;ENDFOLD
      CASE 64
         ;FOLD SPS_TRIG64{H}
         ;ENDFOLD
      CASE 65
         ;FOLD SPS_TRIG65{H}
         ;ENDFOLD
      CASE 66
         ;FOLD SPS_TRIG66{H}
         ;ENDFOLD
      CASE 67
         ;FOLD SPS_TRIG67{H}
         ;ENDFOLD
      CASE 68
         ;FOLD SPS_TRIG68{H}
         ;ENDFOLD
      CASE 69
         ;FOLD SPS_TRIG69{H}
         ;ENDFOLD
      CASE 70
         ;FOLD SPS_TRIG70{H}
         ;ENDFOLD
      CASE 71
         ;FOLD SPS_TRIG71{H}
         ;ENDFOLD
      CASE 72
         ;FOLD SPS_TRIG72{H}
         ;ENDFOLD
      CASE 73
         ;FOLD SPS_TRIG73{H}
         ;ENDFOLD
      CASE 74
         ;FOLD SPS_TRIG74{H}
         ;ENDFOLD
      CASE 75
         ;FOLD SPS_TRIG75{H}
         ;ENDFOLD
      CASE 76
         ;FOLD SPS_TRIG76{H}
         ;ENDFOLD
      CASE 77
         ;FOLD SPS_TRIG77{H}
         ;ENDFOLD
      CASE 78
         ;FOLD SPS_TRIG78{H}
         ;ENDFOLD
      CASE 79
         ;FOLD SPS_TRIG79{H}
         ;ENDFOLD
      CASE 80
         ;FOLD SPS_TRIG80{H}
         ;ENDFOLD
      CASE 81
         ;FOLD SPS_TRIG81{H}
         ;ENDFOLD
      CASE 82
         ;FOLD SPS_TRIG82{H}
         ;ENDFOLD
      CASE 83
         ;FOLD SPS_TRIG83{H}
         ;ENDFOLD
      CASE 84
         ;FOLD SPS_TRIG84{H}
         ;ENDFOLD
      CASE 85
         ;FOLD SPS_TRIG85{H}
         ;ENDFOLD
      CASE 86
         ;FOLD SPS_TRIG86{H}
         ;ENDFOLD
      CASE 87
         ;FOLD SPS_TRIG87{H}
         ;ENDFOLD
      CASE 88
         ;FOLD SPS_TRIG88{H}
         ;ENDFOLD
      CASE 89
         ;FOLD SPS_TRIG89{H}
         ;ENDFOLD
      CASE 90
         ;FOLD SPS_TRIG90{H}
         ;ENDFOLD
      CASE 91
         ;FOLD SPS_TRIG91{H}
         ;ENDFOLD
      CASE 92
         ;FOLD SPS_TRIG92{H}
         ;ENDFOLD
      CASE 93
         ;FOLD SPS_TRIG93{H}
         ;ENDFOLD
      CASE 94
         ;FOLD SPS_TRIG94{H}
         ;ENDFOLD
      CASE 95
         ;FOLD SPS_TRIG95{H}
         ;ENDFOLD
      CASE 96
         ;FOLD SPS_TRIG96{H}
         ;ENDFOLD
      CASE 97
         ;FOLD SPS_TRIG97{H}
         ;ENDFOLD
      CASE 98
         ;FOLD SPS_TRIG98{H}
         ;ENDFOLD
      CASE 99
         ;FOLD SPS_TRIG99{H}
         ;ENDFOLD
      CASE 100
         ;FOLD SPS_TRIG100{H}
         ;ENDFOLD
      CASE 101
         ;FOLD SPS_TRIG101{H}
         ;ENDFOLD
      CASE 102
         ;FOLD SPS_TRIG102{H}
         ;ENDFOLD
      CASE 103
         ;FOLD SPS_TRIG103{H}
         ;ENDFOLD
      CASE 104
         ;FOLD SPS_TRIG104{H}
         ;ENDFOLD
      CASE 105
         ;FOLD SPS_TRIG105{H}
         ;ENDFOLD
      CASE 106
         ;FOLD SPS_TRIG106{H}
         ;ENDFOLD
      CASE 107
         ;FOLD SPS_TRIG107{H}
         ;ENDFOLD
      CASE 108
         ;FOLD SPS_TRIG108{H}
         ;ENDFOLD
      CASE 109
         ;FOLD SPS_TRIG109{H}
         ;ENDFOLD
      CASE 110
         ;FOLD SPS_TRIG110{H}
         ;ENDFOLD
      CASE 111
         ;FOLD SPS_TRIG111{H}
         ;ENDFOLD
      CASE 112
         ;FOLD SPS_TRIG112{H}
         ;ENDFOLD
      CASE 113
         ;FOLD SPS_TRIG113{H}
         ;ENDFOLD
      CASE 114
         ;FOLD SPS_TRIG114{H}
         ;ENDFOLD
      CASE 115
         ;FOLD SPS_TRIG115{H}
         ;ENDFOLD
      CASE 116
         ;FOLD SPS_TRIG116{H}
         ;ENDFOLD
      CASE 117
         ;FOLD SPS_TRIG117{H}
         ;ENDFOLD
      CASE 118
         ;FOLD SPS_TRIG118{H}
         ;ENDFOLD
      CASE 119
         ;FOLD SPS_TRIG119{H}
         ;ENDFOLD
      CASE 120
         ;FOLD SPS_TRIG120{H}
         ;ENDFOLD
      CASE 121
         ;FOLD SPS_TRIG121{H}
         ;ENDFOLD
      CASE 122
         ;FOLD SPS_TRIG122{H}
         ;ENDFOLD
      CASE 123
         ;FOLD SPS_TRIG123{H}
         ;ENDFOLD
      CASE 124
         ;FOLD SPS_TRIG124{H}
         ;ENDFOLD
      CASE 125
         ;FOLD SPS_TRIG125{H}
         ;ENDFOLD
      CASE 126
         ;FOLD SPS_TRIG126{H}
         ;ENDFOLD
      CASE 127
         ;FOLD SPS_TRIG127{H}
         ;ENDFOLD
   DEFAULT
   ENDSWITCH
   ; FOLD ;%{H}
   IF ($MODE_OP<>#EX) THEN
      ;-- Trigger erst nach Wiederanstart geschaltet --
      IF ((((VW_STOP B_AND 'B10010') >0) AND ((VW_STOP B_AND 'B0001')<=0))) THEN
         ;-- MStep Bewegung --
         HALT
      ENDIF
   ENDIF
   ; ENDFOLD
   IF NOT UES THEN
      SPS_FERTIG=TRUE
   ENDIF
END
; ENDFOLD

--- Up86.dat ---
&ACCESS RVP
&REL 328
&COMMENT Abdocken 380 Andocken 379
&PARAM DISKPATH = KRC:\R1\UPs
&PARAM TEMPLATE = C:\KRC\Roboter\Template\upvorgabe
&PARAM EDITMASK = Up999[1-999]
&PARAM TPVW_VERSION = 8.1.8
DEFDAT UP86
; FOLD ;%{H} %MKUKATPVW
; ENDFOLD
; interface to basic routines
 EXT  BAS (BAS_COMMAND  :IN,REAL  :IN )
; interface to VW-standard routines
EXT VW (VW_COMMAND:IN, BOOL: IN, REAL:IN, REAL:IN, REAL:IN, REAL:IN, BOOL :IN, E6POS :IN )
; interface to VW_USER - Call
EXT  VW_USER (VW_USER_CMD :IN,INT :IN,REAL  :IN,REAL  :IN,REAL  :IN,REAL  :IN,REAL  :IN,REAL  :IN,BOOL  :IN )
EXT  VW_USR_R (VW_USER_CMD :IN,INT :IN,REAL  :IN,REAL  :IN,REAL  :IN,REAL  :IN,REAL  :IN,REAL  :IN,BOOL  :IN )
EXT  IBGN (IBGN_COMMAND  :IN,BOOL  :IN,REAL  :IN,REAL  :IN,BOOL  :IN,E6POS  :OUT )
; interface select routine
EXTFCT INT  SELECT (SUBTYPE  :IN,INT  :IN,BOOL  :IN,ARI_TYP  :IN,INT  :IN,BOOL_TYP  :IN,INT  :IN,BOOL  :IN)
INT VW_NEXT_FREE = 27
INT VW_NFREE_SPS = 27
INT VW_MAX_SPS = 127
DECL VW_MPARA_TYP P1_D = {TOOL_NO 32,BASE_NO 0,VB 100,VE 0,ACC 100,TRG_TIME 0,MOVE_TYPE #PTP_MOTION}
DECL E6POS P1 = {X 1080.68, Y -444.7422, Z 2276.944, A 0.003799805, B 29.99818, C -89.99588, S 2, T 42 , E1 0.0, E2 0.0, E3 0.0, E4 0.0, E5 0.0, E6 0.0}
DECL VW_MPARA_TYP P2_D = {TOOL_NO 32,BASE_NO 0,VB 100,VE 100,ACC 100,TRG_TIME 0,MOVE_TYPE #PTP_MOTION}
DECL E6POS P2 = {X 1478.024, Y -384.0801, Z 1627.936, A 16.59922, B 65.89522, C 24.32238, S 2, T 42 , E1 0.0, E2 0.0, E3 0.0, E4 0.0, E5 0.0, E6 0.0}
DECL VW_MPARA_TYP P3_D = {TOOL_NO 32,BASE_NO 0,VB 100,VE 100,ACC 100,TRG_TIME 0,MOVE_TYPE #PTP_MOTION}
DECL E6POS P3 = {X 1076.818, Y -770.2963, Z 693.4174, A 144.5881, B 79.59711, C 137.2426, S 2, T 34 , E1 0.0, E2 0.0, E3 0.0, E4 0.0, E5 0.0, E6 0.0}
DECL VW_MPARA_TYP P4_D = {TOOL_NO 32,BASE_NO 0,VB 100,VE 100,ACC 100,TRG_TIME 0,MOVE_TYPE #PTP_MOTION}
DECL E6POS P4 = {X 1011.646, Y -770.2955, Z 53.22867, A 144.5861, B 79.5973, C 137.2452, S 2, T 34 , E1 0.0, E2 0.0, E3 0.0, E4 0.0, E5 0.0, E6 0.0}
DECL VW_MPARA_TYP P5_D = {TOOL_NO 32,BASE_NO 0,VB 100,VE 100,ACC 100,TRG_TIME 0,MOVE_TYPE #PTP_MOTION}
DECL E6POS P5 = {X 914.1562, Y -628.2295, Z -86.19533, A -28.56616, B 89.61681, C -26.67244, S 6, T 50 , E1 0.0, E2 0.0, E3 0.0, E4 0.0, E5 0.0, E6 0.0}
DECL VW_MPARA_TYP P6_D = {TOOL_NO 32,BASE_NO 0,VB 100,VE 0,ACC 100,TRG_TIME 0,MOVE_TYPE #PTP_MOTION}
DECL E6POS P6 = {X 916.024, Y -629.2413, Z -404.6991, A -28.49056, B 89.61744, C -26.60618, S 6, T 50 , E1 0.0, E2 0.0, E3 0.0, E4 0.0, E5 0.0, E6 0.0}
DECL VW_MPARA_TYP P7_D = {TOOL_NO 32,BASE_NO 0,VB 200,VE 0,ACC 100,TRG_TIME 5,MOVE_TYPE #PATH_MOTION}
DECL E6POS P7 = {X 916.2007, Y -629.3368, Z -434.6989, A -28.49269, B 89.61742, C -26.60826, S 6, T 50 , E1 0.0, E2 0.0, E3 0.0, E4 0.0, E5 0.0, E6 0.0}
DECL VW_MPARA_TYP P8_D = {TOOL_NO 32,BASE_NO 0,VB 50,VE 0,ACC 100,TRG_TIME 5,MOVE_TYPE #PATH_MOTION}
DECL E6POS P8 = {X 916.3768, Y -629.4324, Z -464.699, A -28.49341, B 89.61742, C -26.60887, S 6, T 50 , E1 0.0, E2 0.0, E3 0.0, E4 0.0, E5 0.0, E6 0.0}
DECL VW_MPARA_TYP P9_D = {TOOL_NO 32,BASE_NO 0,VB 50,VE 10,ACC 100,TRG_TIME 5,MOVE_TYPE #PATH_MOTION}
DECL E6POS P9 = {X 916.2006, Y -629.3366, Z -434.6989, A -28.49216, B 89.61743, C -26.60772, S 6, T 50 , E1 0.0, E2 0.0, E3 0.0, E4 0.0, E5 0.0, E6 0.0}
DECL VW_MPARA_TYP P10_D = {TOOL_NO 32,BASE_NO 0,VB 100,VE 50,ACC 100,TRG_TIME 0,MOVE_TYPE #PATH_MOTION}
DECL E6POS P10 = {X 916.0245, Y -629.2414, Z -404.6991, A -28.491, B 89.61741, C -26.60662, S 6, T 50 , E1 0.0, E2 0.0, E3 0.0, E4 0.0, E5 0.0, E6 0.0}
DECL VW_MPARA_TYP P11_D = {TOOL_NO 32,BASE_NO 0,VB 100,VE 100,ACC 100,TRG_TIME 0,MOVE_TYPE #PTP_MOTION}
DECL E6POS P11 = {X 918.4966, Y -631.1271, Z -186.9937, A -28.4373, B 89.6168, C -26.54389, S 6, T 50 , E1 0.0, E2 0.0, E3 0.0, E4 0.0, E5 0.0, E6 0.0}
DECL VW_MPARA_TYP P12_D = {TOOL_NO 32,BASE_NO 0,VB 100,VE 100,ACC 100,TRG_TIME 0,MOVE_TYPE #PTP_MOTION}
DECL E6POS P12 = {X 1300.542, Y -1400.828, Z 103.8305, A -79.95998, B 86.99388, C -103.6366, S 2, T 34 , E1 0.0, E2 0.0, E3 0.0, E4 0.0, E5 0.0, E6 0.0}
DECL VW_MPARA_TYP P13_D = {TOOL_NO 32,BASE_NO 0,VB 100,VE 0,ACC 100,TRG_TIME 0,MOVE_TYPE #PTP_MOTION}
DECL E6POS P13 = {X 1300.542, Y -1400.827, Z 103.8304, A -79.96008, B 86.99389, C -103.6367, S 2, T 34 , E1 0.0, E2 0.0, E3 0.0, E4 0.0, E5 0.0, E6 0.0}
DECL VW_MPARA_TYP P14_D = {TOOL_NO 32,BASE_NO 0,VB 100,VE 0,ACC 100,TRG_TIME 0,MOVE_TYPE #PTP_MOTION}
DECL E6POS P14 = {X 1339.442, Y -1322.11, Z 101.0398, A -130.8366, B 5.095043, C 88.68829, S 2, T 34 , E1 0.0, E2 0.0, E3 0.0, E4 0.0, E5 0.0, E6 0.0}
DECL VW_MPARA_TYP P15_D = {TOOL_NO 32,BASE_NO 0,VB 100,VE 0,ACC 100,TRG_TIME 0,MOVE_TYPE #PTP_MOTION}
DECL E6POS P15 = {X 1300.545, Y -1400.827, Z 103.8308, A -79.95303, B 86.99385, C -103.6299, S 2, T 34 , E1 0.0, E2 0.0, E3 0.0, E4 0.0, E5 0.0, E6 0.0}
DECL VW_MPARA_TYP P16_D = {TOOL_NO 32,BASE_NO 0,VB 100,VE 100,ACC 100,TRG_TIME 0,MOVE_TYPE #PTP_MOTION}
DECL E6POS P16 = {X 1597.213, Y -2278.041, Z -58.6368, A 22.07564, B 89.5185, C 4.188063, S 2, T 42 , E1 0.0, E2 0.0, E3 0.0, E4 0.0, E5 0.0, E6 0.0}
DECL VW_MPARA_TYP P17_D = {TOOL_NO 32,BASE_NO 0,VB 100,VE 100,ACC 100,TRG_TIME 0,MOVE_TYPE #PTP_MOTION}
DECL E6POS P17 = {X 1598.493, Y -2277.579, Z -203.375, A 22.10468, B 89.51871, C 4.359868, S 2, T 42 , E1 0.0, E2 0.0, E3 0.0, E4 0.0, E5 0.0, E6 0.0}
DECL VW_MPARA_TYP P18_D = {TOOL_NO 32,BASE_NO 0,VB 300,VE 0,ACC 100,TRG_TIME 5,MOVE_TYPE #PATH_MOTION}
DECL E6POS P18 = {X 1598.729, Y -2277.483, Z -233.3748, A 22.10886, B 89.51855, C 4.364119, S 2, T 42 , E1 0.0, E2 0.0, E3 0.0, E4 0.0, E5 0.0, E6 0.0}
DECL VW_MPARA_TYP P19_D = {TOOL_NO 32,BASE_NO 0,VB 100,VE 0,ACC 100,TRG_TIME 5,MOVE_TYPE #PATH_MOTION}
DECL E6POS P19 = {X 1598.979, Y -2277.382, Z -265.5069, A 22.09669, B 89.51857, C 4.351958, S 2, T 42 , E1 0.0, E2 0.0, E3 0.0, E4 0.0, E5 0.0, E6 0.0}
DECL VW_MPARA_TYP P20_D = {TOOL_NO 32,BASE_NO 0,VB 50,VE 0,ACC 100,TRG_TIME 5,MOVE_TYPE #PATH_MOTION}
DECL E6POS P20 = {X 1598.729, Y -2277.483, Z -233.3747, A 22.10732, B 89.51855, C 4.36259, S 2, T 42 , E1 0.0, E2 0.0, E3 0.0, E4 0.0, E5 0.0, E6 0.0}
DECL VW_MPARA_TYP P21_D = {TOOL_NO 32,BASE_NO 0,VB 200,VE 10,ACC 100,TRG_TIME 0,MOVE_TYPE #PATH_MOTION}
DECL E6POS P21 = {X 1598.603, Y -2277.525, Z -219.9444, A 22.18919, B 89.51914, C 4.443736, S 2, T 42 , E1 0.0, E2 0.0, E3 0.0, E4 0.0, E5 0.0, E6 0.0}
DECL VW_MPARA_TYP P22_D = {TOOL_NO 32,BASE_NO 0,VB 800,VE 100,ACC 100,TRG_TIME 0,MOVE_TYPE #PATH_MOTION}
DECL E6POS P22 = {X 1519.143, Y -2302.957, Z -220.6371, A 22.17651, B 89.51916, C 4.429426, S 2, T 42 , E1 0.0, E2 0.0, E3 0.0, E4 0.0, E5 0.0, E6 0.0}
DECL VW_MPARA_TYP P23_D = {TOOL_NO 32,BASE_NO 0,VB 100,VE 100,ACC 100,TRG_TIME 0,MOVE_TYPE #PTP_MOTION}
DECL E6POS P23 = {X 1551.986, Y -2352.849, Z 283.0602, A -53.67625, B 80.84645, C -71.46075, S 2, T 42 , E1 0.0, E2 0.0, E3 0.0, E4 0.0, E5 0.0, E6 0.0}
DECL VW_MPARA_TYP P24_D = {TOOL_NO 32,BASE_NO 0,VB 100,VE 100,ACC 100,TRG_TIME 0,MOVE_TYPE #PTP_MOTION}
DECL E6POS P24 = {X 1699.837, Y -2248.959, Z 1063.911, A -51.93394, B 62.88195, C -73.46794, S 2, T 42 , E1 0.0, E2 0.0, E3 0.0, E4 0.0, E5 0.0, E6 0.0}
DECL VW_MPARA_TYP P25_D = {TOOL_NO 32,BASE_NO 0,VB 100,VE 100,ACC 100,TRG_TIME 0,MOVE_TYPE #PTP_MOTION}
DECL E6POS P25 = {X 1661.622, Y -1781.202, Z 1759.068, A -38.57869, B 50.31991, C -63.2539, S 2, T 42 , E1 0.0, E2 0.0, E3 0.0, E4 0.0, E5 0.0, E6 0.0}
DECL VW_MPARA_TYP P26_D = {TOOL_NO 32,BASE_NO 0,VB 100,VE 0,ACC 100,TRG_TIME 0,MOVE_TYPE #PTP_MOTION}
DECL E6POS P26 = {X 1080.68, Y -444.7421, Z 2276.944, A 0.003816008, B 29.99818, C -89.99586, S 2, T 42 , E1 0.0, E2 0.0, E3 0.0, E4 0.0, E5 0.0, E6 0.0}
ENDDAT
